REGION Network 60: ST04->ST05
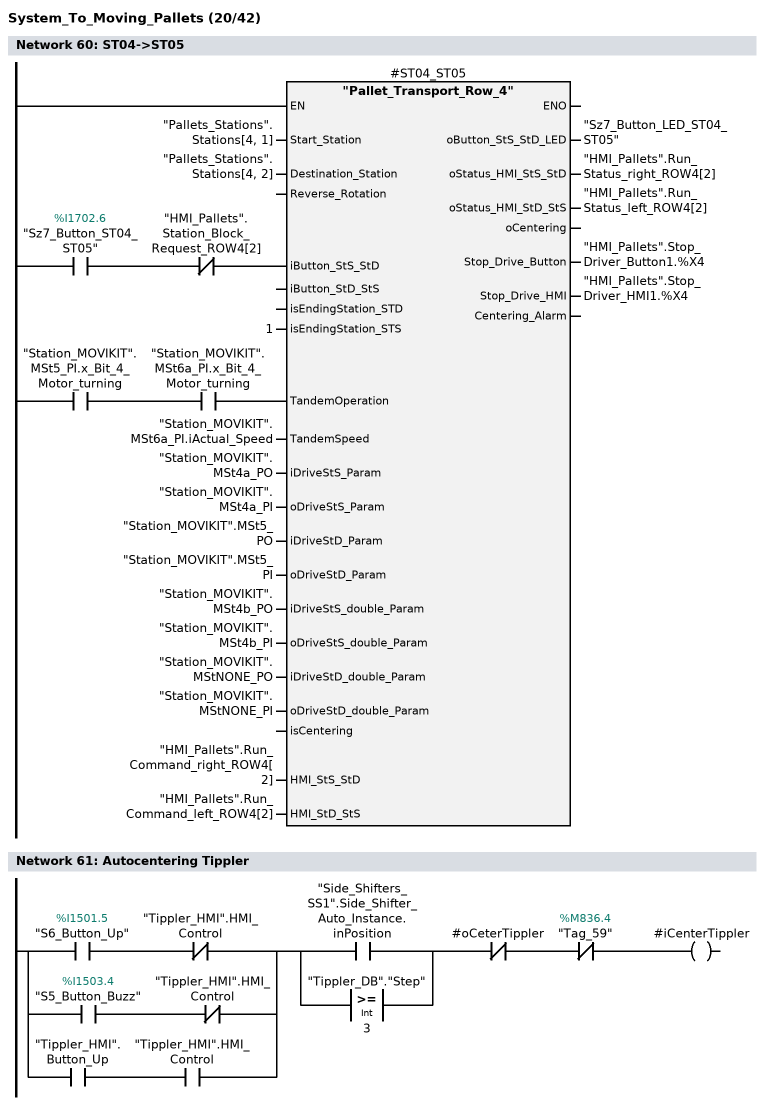
   RUNG wire#powerrail
      #ST04_ST05(iButton_StS_StD := wire#w1, TandemOperation := wire#w2, Start_Station := "Pallets_Stations".Stations[4, 1], Destination_Station := "Pallets_Stations".Stations[4, 2], Reverse_Rotation :=, iButton_StD_StS :=, isEndingStation_STD :=, isEndingStation_STS := 1, TandemSpeed := "Station_MOVIKIT".MSt6a_PI.iActual_Speed, iDriveStS_Param := "Station_MOVIKIT".MSt4a_PO, oDriveStS_Param := "Station_MOVIKIT".MSt4a_PI, iDriveStD_Param := "Station_MOVIKIT".MSt5_PO, oDriveStD_Param := "Station_MOVIKIT".MSt5_PI, iDriveStS_double_Param := "Station_MOVIKIT".MSt4b_PO, oDriveStS_double_Param := "Station_MOVIKIT".MSt4b_PI, iDriveStD_double_Param := "Station_MOVIKIT".MStNONE_PO, oDriveStD_double_Param := "Station_MOVIKIT".MStNONE_PI, isCentering :=, HMI_StS_StD := "HMI_Pallets".Run_Command_right_ROW4[2], HMI_StD_StS := "HMI_Pallets".Run_Command_left_ROW4[2], oButton_StS_StD_LED => "Sz7_Button_LED_ST04_ST05", oStatus_HMI_StS_StD => "HMI_Pallets".Run_Status_right_ROW4[2], oStatus_HMI_StD_StS => "HMI_Pallets".Run_Status_left_ROW4[2], oCentering =>, Stop_Drive_Button => "HMI_Pallets".Stop_Driver_Button1.%X4, Stop_Drive_HMI => "HMI_Pallets".Stop_Driver_HMI1.%X4, Centering_Alarm =>)
   END_RUNG
   RUNG wire#powerrail
      Contact( "Sz7_Button_ST04_ST05" )
      I_Contact( "HMI_Pallets".Station_Block_Request_ROW4[2] )
   END_RUNG wire#w1
   RUNG wire#powerrail
      Contact( "Station_MOVIKIT".MSt5_PI.x_Bit_4_Motor_turning )
      Contact( "Station_MOVIKIT".MSt6a_PI.x_Bit_4_Motor_turning )
   END_RUNG wire#w2
   // the same network as SCL:
   #ST04_ST05(Start_Station := "Pallets_Stations".Stations[4, 1],   // "Pallet_Transport_Row_4"
              Destination_Station := "Pallets_Stations".Stations[4, 2],
              iButton_StS_StD := "Sz7_Button_ST04_ST05" AND NOT "HMI_Pallets".Station_Block_Request_ROW4[2],
              isEndingStation_STS := 1,
              TandemOperation := "Station_MOVIKIT".MSt5_PI.x_Bit_4_Motor_turning AND "Station_MOVIKIT".MSt6a_PI.x_Bit_4_Motor_turning,
              TandemSpeed := "Station_MOVIKIT".MSt6a_PI.iActual_Speed,
              iDriveStS_Param := "Station_MOVIKIT".MSt4a_PO,
              oDriveStS_Param := "Station_MOVIKIT".MSt4a_PI,
              iDriveStD_Param := "Station_MOVIKIT".MSt5_PO,
              oDriveStD_Param := "Station_MOVIKIT".MSt5_PI,
              iDriveStS_double_Param := "Station_MOVIKIT".MSt4b_PO,
              oDriveStS_double_Param := "Station_MOVIKIT".MSt4b_PI,
              iDriveStD_double_Param := "Station_MOVIKIT".MStNONE_PO,
              oDriveStD_double_Param := "Station_MOVIKIT".MStNONE_PI,
              HMI_StS_StD := "HMI_Pallets".Run_Command_right_ROW4[2],
              HMI_StD_StS := "HMI_Pallets".Run_Command_left_ROW4[2],
              oButton_StS_StD_LED => "Sz7_Button_LED_ST04_ST05",
              oStatus_HMI_StS_StD => "HMI_Pallets".Run_Status_right_ROW4[2],
              oStatus_HMI_StD_StS => "HMI_Pallets".Run_Status_left_ROW4[2],
              Stop_Drive_Button => "HMI_Pallets".Stop_Driver_Button1.%X4,
              Stop_Drive_HMI => "HMI_Pallets".Stop_Driver_HMI1.%X4);
END_REGION

REGION Network 61: Autocentering Tippler
   RUNG wire#powerrail
      Contact( "S6_Button_Up" )
      I_Contact( "Tippler_HMI".HMI_Control )
      wire#w1
      Contact( "Side_Shifters_SS1".Side_Shifter_Auto_Instance.inPosition )
      wire#w2
      I_Contact( #oCeterTippler )
      I_Contact( "Tag_59" )
      Coil( #iCenterTippler )
   END_RUNG
   RUNG wire#powerrail
      Contact( "S5_Button_Buzz" )
      I_Contact( "Tippler_HMI".HMI_Control )
   END_RUNG wire#w1
   RUNG wire#powerrail
      Contact( "Tippler_HMI".Button_Up )
      Contact( "Tippler_HMI".HMI_Control )
   END_RUNG wire#w1
   RUNG wire#w1
      { S7_Templates := "SrcType := Int" } GE_Contact(in1 := "Tippler_DB"."Step", in2 := 3)
   END_RUNG wire#w2
   // the same network as SCL:
   #iCenterTippler := (("S6_Button_Up" AND NOT "Tippler_HMI".HMI_Control) OR ("S5_Button_Buzz" AND NOT "Tippler_HMI".HMI_Control) OR ("Tippler_HMI".Button_Up AND "Tippler_HMI".HMI_Control)) AND ("Side_Shifters_SS1".Side_Shifter_Auto_Instance.inPosition OR ("Tippler_DB"."Step" >= 3)) AND NOT #oCeterTippler AND NOT "Tag_59";
END_REGION

REGION Network 62: ST01->ST02
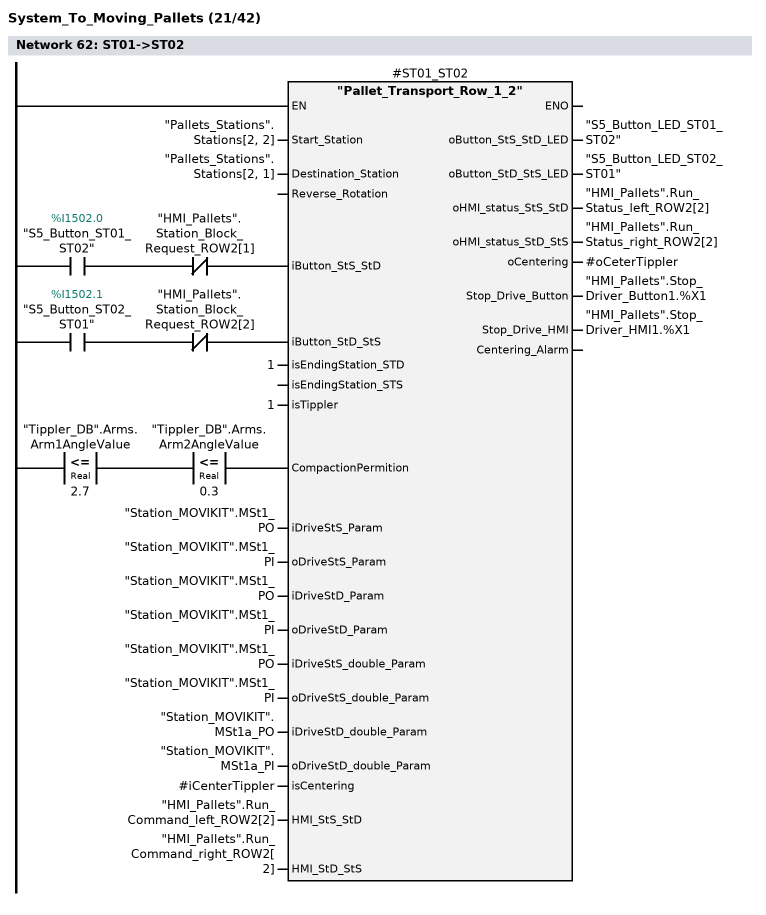
   RUNG wire#powerrail
      #ST01_ST02(iButton_StS_StD := wire#w1, iButton_StD_StS := wire#w2, CompactionPermition := wire#w3, Start_Station := "Pallets_Stations".Stations[2, 2], Destination_Station := "Pallets_Stations".Stations[2, 1], Reverse_Rotation :=, isEndingStation_STD := 1, isEndingStation_STS :=, isTippler := 1, iDriveStS_Param := "Station_MOVIKIT".MSt1_PO, oDriveStS_Param := "Station_MOVIKIT".MSt1_PI, iDriveStD_Param := "Station_MOVIKIT".MSt1_PO, oDriveStD_Param := "Station_MOVIKIT".MSt1_PI, iDriveStS_double_Param := "Station_MOVIKIT".MSt1_PO, oDriveStS_double_Param := "Station_MOVIKIT".MSt1_PI, iDriveStD_double_Param := "Station_MOVIKIT".MSt1a_PO, oDriveStD_double_Param := "Station_MOVIKIT".MSt1a_PI, isCentering := #iCenterTippler, HMI_StS_StD := "HMI_Pallets".Run_Command_left_ROW2[2], HMI_StD_StS := "HMI_Pallets".Run_Command_right_ROW2[2], oButton_StS_StD_LED => "S5_Button_LED_ST01_ST02", oButton_StD_StS_LED => "S5_Button_LED_ST02_ST01", oHMI_status_StS_StD => "HMI_Pallets".Run_Status_left_ROW2[2], oHMI_status_StD_StS => "HMI_Pallets".Run_Status_right_ROW2[2], oCentering => #oCeterTippler, Stop_Drive_Button => "HMI_Pallets".Stop_Driver_Button1.%X1, Stop_Drive_HMI => "HMI_Pallets".Stop_Driver_HMI1.%X1, Centering_Alarm =>)
   END_RUNG
   RUNG wire#powerrail
      Contact( "S5_Button_ST01_ST02" )
      I_Contact( "HMI_Pallets".Station_Block_Request_ROW2[1] )
   END_RUNG wire#w1
   RUNG wire#powerrail
      Contact( "S5_Button_ST02_ST01" )
      I_Contact( "HMI_Pallets".Station_Block_Request_ROW2[2] )
   END_RUNG wire#w2
   RUNG wire#powerrail
      { S7_Templates := "SrcType := Real" } LE_Contact(in1 := "Tippler_DB".Arms.Arm1AngleValue, in2 := 2.7)
      { S7_Templates := "SrcType := Real" } LE_Contact(in1 := "Tippler_DB".Arms.Arm2AngleValue, in2 := 0.3)
   END_RUNG wire#w3
   // the same network as SCL:
   #ST01_ST02(Start_Station := "Pallets_Stations".Stations[2, 2],   // "Pallet_Transport_Row_1_2"
              Destination_Station := "Pallets_Stations".Stations[2, 1],
              iButton_StS_StD := "S5_Button_ST01_ST02" AND NOT "HMI_Pallets".Station_Block_Request_ROW2[1],
              iButton_StD_StS := "S5_Button_ST02_ST01" AND NOT "HMI_Pallets".Station_Block_Request_ROW2[2],
              isEndingStation_STD := 1,
              isTippler := 1,
              CompactionPermition := ("Tippler_DB".Arms.Arm1AngleValue <= 2.7) AND ("Tippler_DB".Arms.Arm2AngleValue <= 0.3),
              iDriveStS_Param := "Station_MOVIKIT".MSt1_PO,
              oDriveStS_Param := "Station_MOVIKIT".MSt1_PI,
              iDriveStD_Param := "Station_MOVIKIT".MSt1_PO,
              oDriveStD_Param := "Station_MOVIKIT".MSt1_PI,
              iDriveStS_double_Param := "Station_MOVIKIT".MSt1_PO,
              oDriveStS_double_Param := "Station_MOVIKIT".MSt1_PI,
              iDriveStD_double_Param := "Station_MOVIKIT".MSt1a_PO,
              oDriveStD_double_Param := "Station_MOVIKIT".MSt1a_PI,
              isCentering := #iCenterTippler,
              HMI_StS_StD := "HMI_Pallets".Run_Command_left_ROW2[2],
              HMI_StD_StS := "HMI_Pallets".Run_Command_right_ROW2[2],
              oButton_StS_StD_LED => "S5_Button_LED_ST01_ST02",
              oButton_StD_StS_LED => "S5_Button_LED_ST02_ST01",
              oHMI_status_StS_StD => "HMI_Pallets".Run_Status_left_ROW2[2],
              oHMI_status_StD_StS => "HMI_Pallets".Run_Status_right_ROW2[2],
              oCentering => #oCeterTippler,
              Stop_Drive_Button => "HMI_Pallets".Stop_Driver_Button1.%X1,
              Stop_Drive_HMI => "HMI_Pallets".Stop_Driver_HMI1.%X1);
END_REGION

REGION Network 63: ST38->ST01
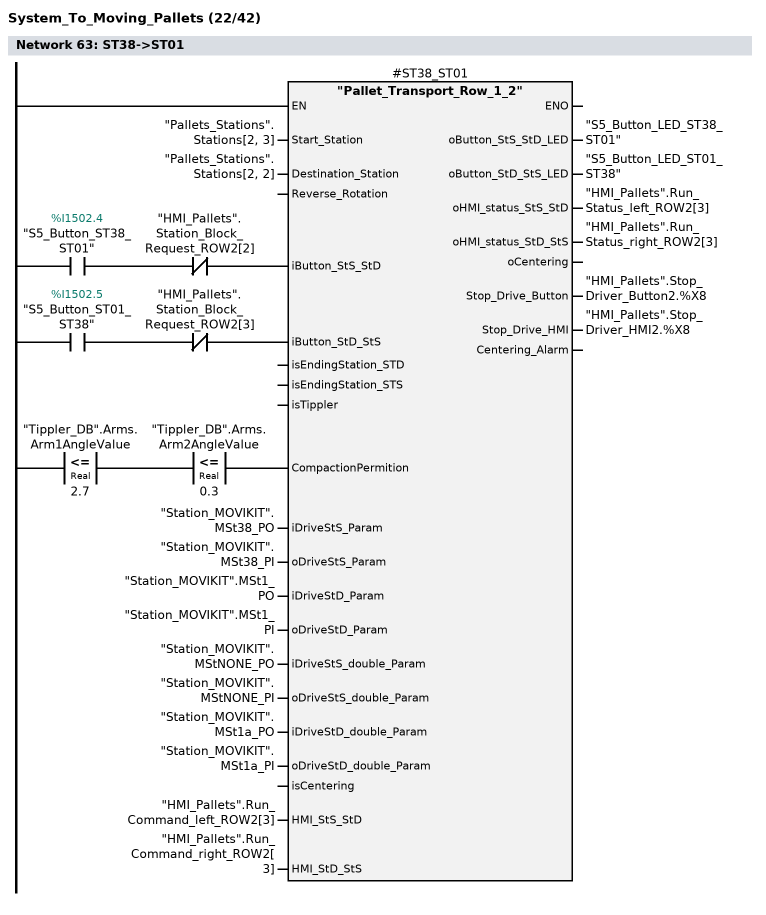
   RUNG wire#powerrail
      #ST38_ST01(iButton_StS_StD := wire#w1, iButton_StD_StS := wire#w2, CompactionPermition := wire#w3, Start_Station := "Pallets_Stations".Stations[2, 3], Destination_Station := "Pallets_Stations".Stations[2, 2], Reverse_Rotation :=, isEndingStation_STD :=, isEndingStation_STS :=, isTippler :=, iDriveStS_Param := "Station_MOVIKIT".MSt38_PO, oDriveStS_Param := "Station_MOVIKIT".MSt38_PI, iDriveStD_Param := "Station_MOVIKIT".MSt1_PO, oDriveStD_Param := "Station_MOVIKIT".MSt1_PI, iDriveStS_double_Param := "Station_MOVIKIT".MStNONE_PO, oDriveStS_double_Param := "Station_MOVIKIT".MStNONE_PI, iDriveStD_double_Param := "Station_MOVIKIT".MSt1a_PO, oDriveStD_double_Param := "Station_MOVIKIT".MSt1a_PI, isCentering :=, HMI_StS_StD := "HMI_Pallets".Run_Command_left_ROW2[3], HMI_StD_StS := "HMI_Pallets".Run_Command_right_ROW2[3], oButton_StS_StD_LED => "S5_Button_LED_ST38_ST01", oButton_StD_StS_LED => "S5_Button_LED_ST01_ST38", oHMI_status_StS_StD => "HMI_Pallets".Run_Status_left_ROW2[3], oHMI_status_StD_StS => "HMI_Pallets".Run_Status_right_ROW2[3], oCentering =>, Stop_Drive_Button => "HMI_Pallets".Stop_Driver_Button2.%X8, Stop_Drive_HMI => "HMI_Pallets".Stop_Driver_HMI2.%X8, Centering_Alarm =>)
   END_RUNG
   RUNG wire#powerrail
      Contact( "S5_Button_ST38_ST01" )
      I_Contact( "HMI_Pallets".Station_Block_Request_ROW2[2] )
   END_RUNG wire#w1
   RUNG wire#powerrail
      Contact( "S5_Button_ST01_ST38" )
      I_Contact( "HMI_Pallets".Station_Block_Request_ROW2[3] )
   END_RUNG wire#w2
   RUNG wire#powerrail
      { S7_Templates := "SrcType := Real" } LE_Contact(in1 := "Tippler_DB".Arms.Arm1AngleValue, in2 := 2.7)
      { S7_Templates := "SrcType := Real" } LE_Contact(in1 := "Tippler_DB".Arms.Arm2AngleValue, in2 := 0.3)
   END_RUNG wire#w3
   // the same network as SCL:
   #ST38_ST01(Start_Station := "Pallets_Stations".Stations[2, 3],   // "Pallet_Transport_Row_1_2"
              Destination_Station := "Pallets_Stations".Stations[2, 2],
              iButton_StS_StD := "S5_Button_ST38_ST01" AND NOT "HMI_Pallets".Station_Block_Request_ROW2[2],
              iButton_StD_StS := "S5_Button_ST01_ST38" AND NOT "HMI_Pallets".Station_Block_Request_ROW2[3],
              CompactionPermition := ("Tippler_DB".Arms.Arm1AngleValue <= 2.7) AND ("Tippler_DB".Arms.Arm2AngleValue <= 0.3),
              iDriveStS_Param := "Station_MOVIKIT".MSt38_PO,
              oDriveStS_Param := "Station_MOVIKIT".MSt38_PI,
              iDriveStD_Param := "Station_MOVIKIT".MSt1_PO,
              oDriveStD_Param := "Station_MOVIKIT".MSt1_PI,
              iDriveStS_double_Param := "Station_MOVIKIT".MStNONE_PO,
              oDriveStS_double_Param := "Station_MOVIKIT".MStNONE_PI,
              iDriveStD_double_Param := "Station_MOVIKIT".MSt1a_PO,
              oDriveStD_double_Param := "Station_MOVIKIT".MSt1a_PI,
              HMI_StS_StD := "HMI_Pallets".Run_Command_left_ROW2[3],
              HMI_StD_StS := "HMI_Pallets".Run_Command_right_ROW2[3],
              oButton_StS_StD_LED => "S5_Button_LED_ST38_ST01",
              oButton_StD_StS_LED => "S5_Button_LED_ST01_ST38",
              oHMI_status_StS_StD => "HMI_Pallets".Run_Status_left_ROW2[3],
              oHMI_status_StD_StS => "HMI_Pallets".Run_Status_right_ROW2[3],
              Stop_Drive_Button => "HMI_Pallets".Stop_Driver_Button2.%X8,
              Stop_Drive_HMI => "HMI_Pallets".Stop_Driver_HMI2.%X8);
END_REGION

REGION Network 64: ST34->ST35
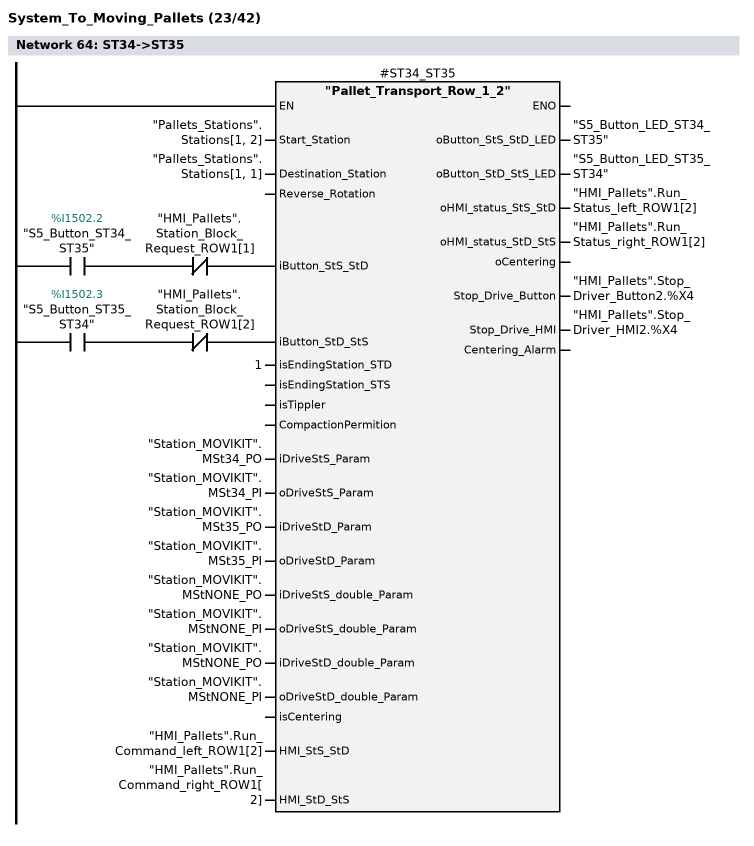
   RUNG wire#powerrail
      #ST34_ST35(iButton_StS_StD := wire#w1, iButton_StD_StS := wire#w2, Start_Station := "Pallets_Stations".Stations[1, 2], Destination_Station := "Pallets_Stations".Stations[1, 1], Reverse_Rotation :=, isEndingStation_STD := 1, isEndingStation_STS :=, isTippler :=, CompactionPermition :=, iDriveStS_Param := "Station_MOVIKIT".MSt34_PO, oDriveStS_Param := "Station_MOVIKIT".MSt34_PI, iDriveStD_Param := "Station_MOVIKIT".MSt35_PO, oDriveStD_Param := "Station_MOVIKIT".MSt35_PI, iDriveStS_double_Param := "Station_MOVIKIT".MStNONE_PO, oDriveStS_double_Param := "Station_MOVIKIT".MStNONE_PI, iDriveStD_double_Param := "Station_MOVIKIT".MStNONE_PO, oDriveStD_double_Param := "Station_MOVIKIT".MStNONE_PI, isCentering :=, HMI_StS_StD := "HMI_Pallets".Run_Command_left_ROW1[2], HMI_StD_StS := "HMI_Pallets".Run_Command_right_ROW1[2], oButton_StS_StD_LED => "S5_Button_LED_ST34_ST35", oButton_StD_StS_LED => "S5_Button_LED_ST35_ST34", oHMI_status_StS_StD => "HMI_Pallets".Run_Status_left_ROW1[2], oHMI_status_StD_StS => "HMI_Pallets".Run_Status_right_ROW1[2], oCentering =>, Stop_Drive_Button => "HMI_Pallets".Stop_Driver_Button2.%X4, Stop_Drive_HMI => "HMI_Pallets".Stop_Driver_HMI2.%X4, Centering_Alarm =>)
   END_RUNG
   RUNG wire#powerrail
      Contact( "S5_Button_ST34_ST35" )
      I_Contact( "HMI_Pallets".Station_Block_Request_ROW1[1] )
   END_RUNG wire#w1
   RUNG wire#powerrail
      Contact( "S5_Button_ST35_ST34" )
      I_Contact( "HMI_Pallets".Station_Block_Request_ROW1[2] )
   END_RUNG wire#w2
   // the same network as SCL:
   #ST34_ST35(Start_Station := "Pallets_Stations".Stations[1, 2],   // "Pallet_Transport_Row_1_2"
              Destination_Station := "Pallets_Stations".Stations[1, 1],
              iButton_StS_StD := "S5_Button_ST34_ST35" AND NOT "HMI_Pallets".Station_Block_Request_ROW1[1],
              iButton_StD_StS := "S5_Button_ST35_ST34" AND NOT "HMI_Pallets".Station_Block_Request_ROW1[2],
              isEndingStation_STD := 1,
              iDriveStS_Param := "Station_MOVIKIT".MSt34_PO,
              oDriveStS_Param := "Station_MOVIKIT".MSt34_PI,
              iDriveStD_Param := "Station_MOVIKIT".MSt35_PO,
              oDriveStD_Param := "Station_MOVIKIT".MSt35_PI,
              iDriveStS_double_Param := "Station_MOVIKIT".MStNONE_PO,
              oDriveStS_double_Param := "Station_MOVIKIT".MStNONE_PI,
              iDriveStD_double_Param := "Station_MOVIKIT".MStNONE_PO,
              oDriveStD_double_Param := "Station_MOVIKIT".MStNONE_PI,
              HMI_StS_StD := "HMI_Pallets".Run_Command_left_ROW1[2],
              HMI_StD_StS := "HMI_Pallets".Run_Command_right_ROW1[2],
              oButton_StS_StD_LED => "S5_Button_LED_ST34_ST35",
              oButton_StD_StS_LED => "S5_Button_LED_ST35_ST34",
              oHMI_status_StS_StD => "HMI_Pallets".Run_Status_left_ROW1[2],
              oHMI_status_StD_StS => "HMI_Pallets".Run_Status_right_ROW1[2],
              Stop_Drive_Button => "HMI_Pallets".Stop_Driver_Button2.%X4,
              Stop_Drive_HMI => "HMI_Pallets".Stop_Driver_HMI2.%X4);
END_REGION

REGION Network 65: ST33->ST34
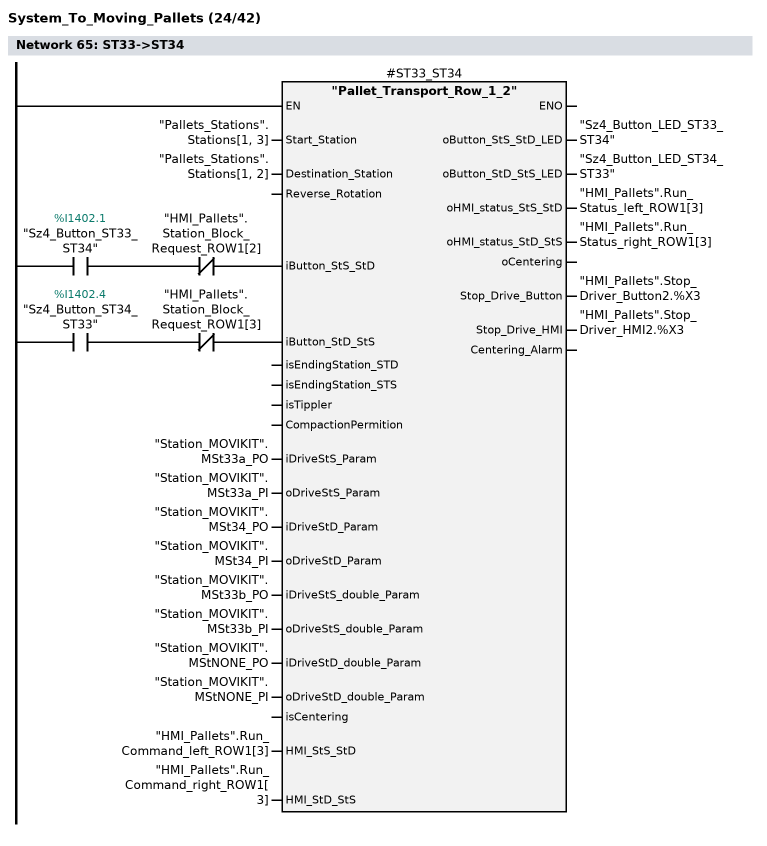
   RUNG wire#powerrail
      #ST33_ST34(iButton_StS_StD := wire#w1, iButton_StD_StS := wire#w2, Start_Station := "Pallets_Stations".Stations[1, 3], Destination_Station := "Pallets_Stations".Stations[1, 2], Reverse_Rotation :=, isEndingStation_STD :=, isEndingStation_STS :=, isTippler :=, CompactionPermition :=, iDriveStS_Param := "Station_MOVIKIT".MSt33a_PO, oDriveStS_Param := "Station_MOVIKIT".MSt33a_PI, iDriveStD_Param := "Station_MOVIKIT".MSt34_PO, oDriveStD_Param := "Station_MOVIKIT".MSt34_PI, iDriveStS_double_Param := "Station_MOVIKIT".MSt33b_PO, oDriveStS_double_Param := "Station_MOVIKIT".MSt33b_PI, iDriveStD_double_Param := "Station_MOVIKIT".MStNONE_PO, oDriveStD_double_Param := "Station_MOVIKIT".MStNONE_PI, isCentering :=, HMI_StS_StD := "HMI_Pallets".Run_Command_left_ROW1[3], HMI_StD_StS := "HMI_Pallets".Run_Command_right_ROW1[3], oButton_StS_StD_LED => "Sz4_Button_LED_ST33_ST34", oButton_StD_StS_LED => "Sz4_Button_LED_ST34_ST33", oHMI_status_StS_StD => "HMI_Pallets".Run_Status_left_ROW1[3], oHMI_status_StD_StS => "HMI_Pallets".Run_Status_right_ROW1[3], oCentering =>, Stop_Drive_Button => "HMI_Pallets".Stop_Driver_Button2.%X3, Stop_Drive_HMI => "HMI_Pallets".Stop_Driver_HMI2.%X3, Centering_Alarm =>)
   END_RUNG
   RUNG wire#powerrail
      Contact( "Sz4_Button_ST33_ST34" )
      I_Contact( "HMI_Pallets".Station_Block_Request_ROW1[2] )
   END_RUNG wire#w1
   RUNG wire#powerrail
      Contact( "Sz4_Button_ST34_ST33" )
      I_Contact( "HMI_Pallets".Station_Block_Request_ROW1[3] )
   END_RUNG wire#w2
   // the same network as SCL:
   #ST33_ST34(Start_Station := "Pallets_Stations".Stations[1, 3],   // "Pallet_Transport_Row_1_2"
              Destination_Station := "Pallets_Stations".Stations[1, 2],
              iButton_StS_StD := "Sz4_Button_ST33_ST34" AND NOT "HMI_Pallets".Station_Block_Request_ROW1[2],
              iButton_StD_StS := "Sz4_Button_ST34_ST33" AND NOT "HMI_Pallets".Station_Block_Request_ROW1[3],
              iDriveStS_Param := "Station_MOVIKIT".MSt33a_PO,
              oDriveStS_Param := "Station_MOVIKIT".MSt33a_PI,
              iDriveStD_Param := "Station_MOVIKIT".MSt34_PO,
              oDriveStD_Param := "Station_MOVIKIT".MSt34_PI,
              iDriveStS_double_Param := "Station_MOVIKIT".MSt33b_PO,
              oDriveStS_double_Param := "Station_MOVIKIT".MSt33b_PI,
              iDriveStD_double_Param := "Station_MOVIKIT".MStNONE_PO,
              oDriveStD_double_Param := "Station_MOVIKIT".MStNONE_PI,
              HMI_StS_StD := "HMI_Pallets".Run_Command_left_ROW1[3],
              HMI_StD_StS := "HMI_Pallets".Run_Command_right_ROW1[3],
              oButton_StS_StD_LED => "Sz4_Button_LED_ST33_ST34",
              oButton_StD_StS_LED => "Sz4_Button_LED_ST34_ST33",
              oHMI_status_StS_StD => "HMI_Pallets".Run_Status_left_ROW1[3],
              oHMI_status_StD_StS => "HMI_Pallets".Run_Status_right_ROW1[3],
              Stop_Drive_Button => "HMI_Pallets".Stop_Driver_Button2.%X3,
              Stop_Drive_HMI => "HMI_Pallets".Stop_Driver_HMI2.%X3);
END_REGION

REGION Network 66: ST32->ST33
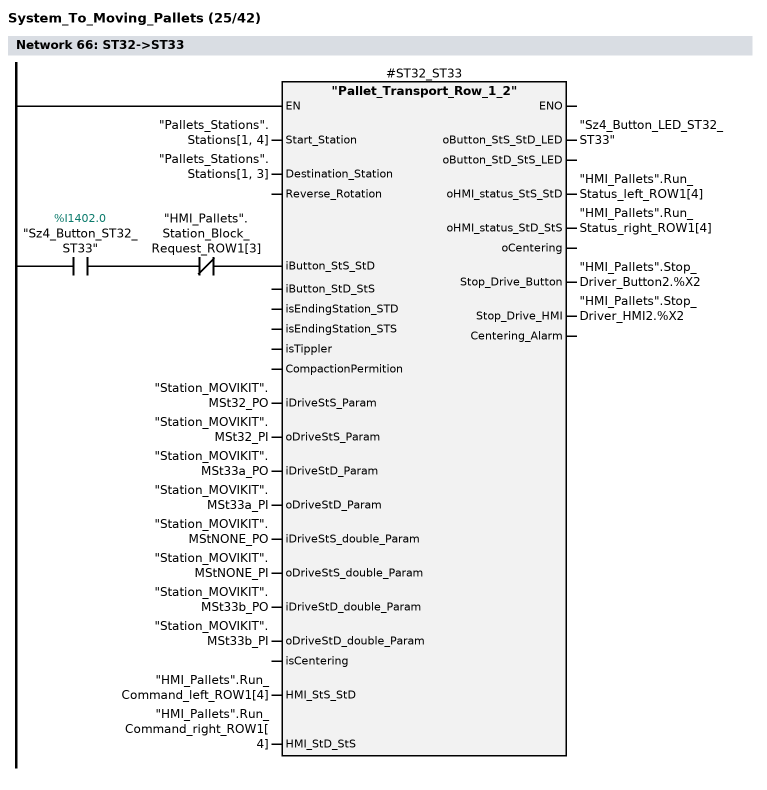
   RUNG wire#powerrail
      #ST32_ST33(iButton_StS_StD := wire#w1, Start_Station := "Pallets_Stations".Stations[1, 4], Destination_Station := "Pallets_Stations".Stations[1, 3], Reverse_Rotation :=, iButton_StD_StS :=, isEndingStation_STD :=, isEndingStation_STS :=, isTippler :=, CompactionPermition :=, iDriveStS_Param := "Station_MOVIKIT".MSt32_PO, oDriveStS_Param := "Station_MOVIKIT".MSt32_PI, iDriveStD_Param := "Station_MOVIKIT".MSt33a_PO, oDriveStD_Param := "Station_MOVIKIT".MSt33a_PI, iDriveStS_double_Param := "Station_MOVIKIT".MStNONE_PO, oDriveStS_double_Param := "Station_MOVIKIT".MStNONE_PI, iDriveStD_double_Param := "Station_MOVIKIT".MSt33b_PO, oDriveStD_double_Param := "Station_MOVIKIT".MSt33b_PI, isCentering :=, HMI_StS_StD := "HMI_Pallets".Run_Command_left_ROW1[4], HMI_StD_StS := "HMI_Pallets".Run_Command_right_ROW1[4], oButton_StS_StD_LED => "Sz4_Button_LED_ST32_ST33", oButton_StD_StS_LED =>, oHMI_status_StS_StD => "HMI_Pallets".Run_Status_left_ROW1[4], oHMI_status_StD_StS => "HMI_Pallets".Run_Status_right_ROW1[4], oCentering =>, Stop_Drive_Button => "HMI_Pallets".Stop_Driver_Button2.%X2, Stop_Drive_HMI => "HMI_Pallets".Stop_Driver_HMI2.%X2, Centering_Alarm =>)
   END_RUNG
   RUNG wire#powerrail
      Contact( "Sz4_Button_ST32_ST33" )
      I_Contact( "HMI_Pallets".Station_Block_Request_ROW1[3] )
   END_RUNG wire#w1
   // the same network as SCL:
   #ST32_ST33(Start_Station := "Pallets_Stations".Stations[1, 4],   // "Pallet_Transport_Row_1_2"
              Destination_Station := "Pallets_Stations".Stations[1, 3],
              iButton_StS_StD := "Sz4_Button_ST32_ST33" AND NOT "HMI_Pallets".Station_Block_Request_ROW1[3],
              iDriveStS_Param := "Station_MOVIKIT".MSt32_PO,
              oDriveStS_Param := "Station_MOVIKIT".MSt32_PI,
              iDriveStD_Param := "Station_MOVIKIT".MSt33a_PO,
              oDriveStD_Param := "Station_MOVIKIT".MSt33a_PI,
              iDriveStS_double_Param := "Station_MOVIKIT".MStNONE_PO,
              oDriveStS_double_Param := "Station_MOVIKIT".MStNONE_PI,
              iDriveStD_double_Param := "Station_MOVIKIT".MSt33b_PO,
              oDriveStD_double_Param := "Station_MOVIKIT".MSt33b_PI,
              HMI_StS_StD := "HMI_Pallets".Run_Command_left_ROW1[4],
              HMI_StD_StS := "HMI_Pallets".Run_Command_right_ROW1[4],
              oButton_StS_StD_LED => "Sz4_Button_LED_ST32_ST33",
              oHMI_status_StS_StD => "HMI_Pallets".Run_Status_left_ROW1[4],
              oHMI_status_StD_StS => "HMI_Pallets".Run_Status_right_ROW1[4],
              Stop_Drive_Button => "HMI_Pallets".Stop_Driver_Button2.%X2,
              Stop_Drive_HMI => "HMI_Pallets".Stop_Driver_HMI2.%X2);
END_REGION

REGION Network 67: ST31->ST32
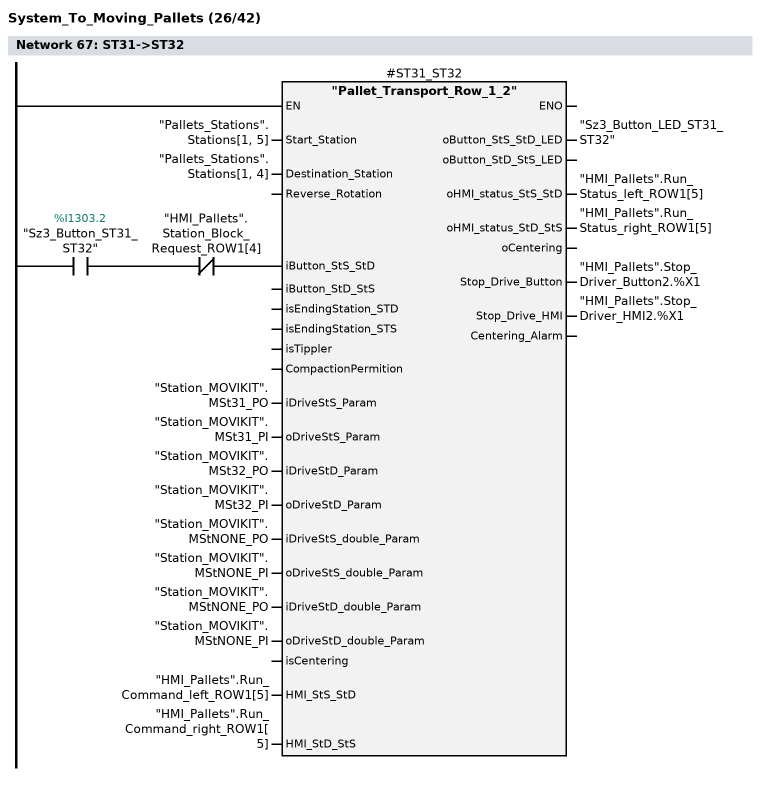
   RUNG wire#powerrail
      #ST31_ST32(iButton_StS_StD := wire#w1, Start_Station := "Pallets_Stations".Stations[1, 5], Destination_Station := "Pallets_Stations".Stations[1, 4], Reverse_Rotation :=, iButton_StD_StS :=, isEndingStation_STD :=, isEndingStation_STS :=, isTippler :=, CompactionPermition :=, iDriveStS_Param := "Station_MOVIKIT".MSt31_PO, oDriveStS_Param := "Station_MOVIKIT".MSt31_PI, iDriveStD_Param := "Station_MOVIKIT".MSt32_PO, oDriveStD_Param := "Station_MOVIKIT".MSt32_PI, iDriveStS_double_Param := "Station_MOVIKIT".MStNONE_PO, oDriveStS_double_Param := "Station_MOVIKIT".MStNONE_PI, iDriveStD_double_Param := "Station_MOVIKIT".MStNONE_PO, oDriveStD_double_Param := "Station_MOVIKIT".MStNONE_PI, isCentering :=, HMI_StS_StD := "HMI_Pallets".Run_Command_left_ROW1[5], HMI_StD_StS := "HMI_Pallets".Run_Command_right_ROW1[5], oButton_StS_StD_LED => "Sz3_Button_LED_ST31_ST32", oButton_StD_StS_LED =>, oHMI_status_StS_StD => "HMI_Pallets".Run_Status_left_ROW1[5], oHMI_status_StD_StS => "HMI_Pallets".Run_Status_right_ROW1[5], oCentering =>, Stop_Drive_Button => "HMI_Pallets".Stop_Driver_Button2.%X1, Stop_Drive_HMI => "HMI_Pallets".Stop_Driver_HMI2.%X1, Centering_Alarm =>)
   END_RUNG
   RUNG wire#powerrail
      Contact( "Sz3_Button_ST31_ST32" )
      I_Contact( "HMI_Pallets".Station_Block_Request_ROW1[4] )
   END_RUNG wire#w1
   // the same network as SCL:
   #ST31_ST32(Start_Station := "Pallets_Stations".Stations[1, 5],   // "Pallet_Transport_Row_1_2"
              Destination_Station := "Pallets_Stations".Stations[1, 4],
              iButton_StS_StD := "Sz3_Button_ST31_ST32" AND NOT "HMI_Pallets".Station_Block_Request_ROW1[4],
              iDriveStS_Param := "Station_MOVIKIT".MSt31_PO,
              oDriveStS_Param := "Station_MOVIKIT".MSt31_PI,
              iDriveStD_Param := "Station_MOVIKIT".MSt32_PO,
              oDriveStD_Param := "Station_MOVIKIT".MSt32_PI,
              iDriveStS_double_Param := "Station_MOVIKIT".MStNONE_PO,
              oDriveStS_double_Param := "Station_MOVIKIT".MStNONE_PI,
              iDriveStD_double_Param := "Station_MOVIKIT".MStNONE_PO,
              oDriveStD_double_Param := "Station_MOVIKIT".MStNONE_PI,
              HMI_StS_StD := "HMI_Pallets".Run_Command_left_ROW1[5],
              HMI_StD_StS := "HMI_Pallets".Run_Command_right_ROW1[5],
              oButton_StS_StD_LED => "Sz3_Button_LED_ST31_ST32",
              oHMI_status_StS_StD => "HMI_Pallets".Run_Status_left_ROW1[5],
              oHMI_status_StD_StS => "HMI_Pallets".Run_Status_right_ROW1[5],
              Stop_Drive_Button => "HMI_Pallets".Stop_Driver_Button2.%X1,
              Stop_Drive_HMI => "HMI_Pallets".Stop_Driver_HMI2.%X1);
END_REGION

REGION Network 68: ST30->ST31
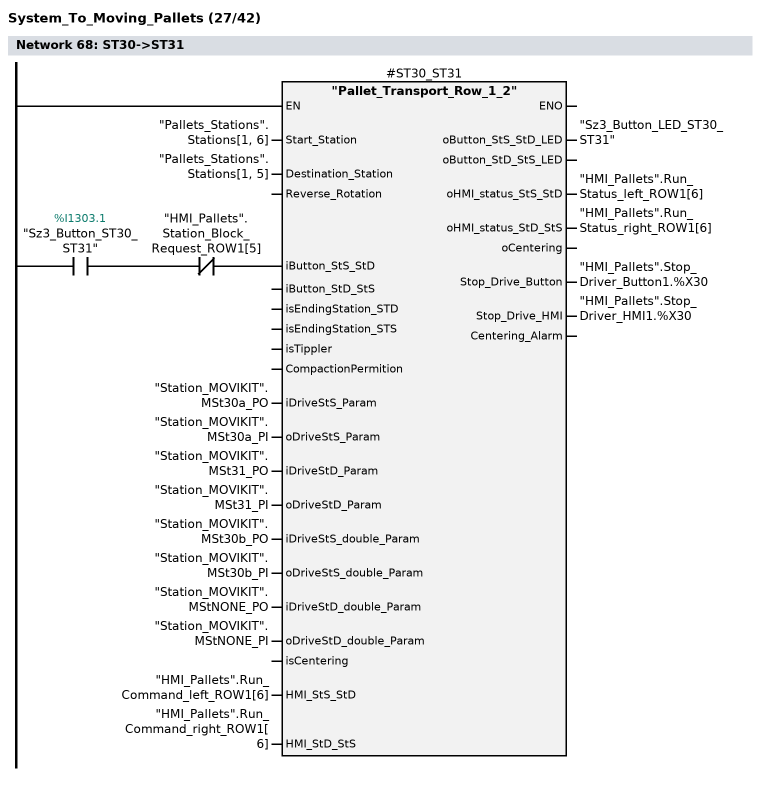
   RUNG wire#powerrail
      #ST30_ST31(iButton_StS_StD := wire#w1, Start_Station := "Pallets_Stations".Stations[1, 6], Destination_Station := "Pallets_Stations".Stations[1, 5], Reverse_Rotation :=, iButton_StD_StS :=, isEndingStation_STD :=, isEndingStation_STS :=, isTippler :=, CompactionPermition :=, iDriveStS_Param := "Station_MOVIKIT".MSt30a_PO, oDriveStS_Param := "Station_MOVIKIT".MSt30a_PI, iDriveStD_Param := "Station_MOVIKIT".MSt31_PO, oDriveStD_Param := "Station_MOVIKIT".MSt31_PI, iDriveStS_double_Param := "Station_MOVIKIT".MSt30b_PO, oDriveStS_double_Param := "Station_MOVIKIT".MSt30b_PI, iDriveStD_double_Param := "Station_MOVIKIT".MStNONE_PO, oDriveStD_double_Param := "Station_MOVIKIT".MStNONE_PI, isCentering :=, HMI_StS_StD := "HMI_Pallets".Run_Command_left_ROW1[6], HMI_StD_StS := "HMI_Pallets".Run_Command_right_ROW1[6], oButton_StS_StD_LED => "Sz3_Button_LED_ST30_ST31", oButton_StD_StS_LED =>, oHMI_status_StS_StD => "HMI_Pallets".Run_Status_left_ROW1[6], oHMI_status_StD_StS => "HMI_Pallets".Run_Status_right_ROW1[6], oCentering =>, Stop_Drive_Button => "HMI_Pallets".Stop_Driver_Button1.%X30, Stop_Drive_HMI => "HMI_Pallets".Stop_Driver_HMI1.%X30, Centering_Alarm =>)
   END_RUNG
   RUNG wire#powerrail
      Contact( "Sz3_Button_ST30_ST31" )
      I_Contact( "HMI_Pallets".Station_Block_Request_ROW1[5] )
   END_RUNG wire#w1
   // the same network as SCL:
   #ST30_ST31(Start_Station := "Pallets_Stations".Stations[1, 6],   // "Pallet_Transport_Row_1_2"
              Destination_Station := "Pallets_Stations".Stations[1, 5],
              iButton_StS_StD := "Sz3_Button_ST30_ST31" AND NOT "HMI_Pallets".Station_Block_Request_ROW1[5],
              iDriveStS_Param := "Station_MOVIKIT".MSt30a_PO,
              oDriveStS_Param := "Station_MOVIKIT".MSt30a_PI,
              iDriveStD_Param := "Station_MOVIKIT".MSt31_PO,
              oDriveStD_Param := "Station_MOVIKIT".MSt31_PI,
              iDriveStS_double_Param := "Station_MOVIKIT".MSt30b_PO,
              oDriveStS_double_Param := "Station_MOVIKIT".MSt30b_PI,
              iDriveStD_double_Param := "Station_MOVIKIT".MStNONE_PO,
              oDriveStD_double_Param := "Station_MOVIKIT".MStNONE_PI,
              HMI_StS_StD := "HMI_Pallets".Run_Command_left_ROW1[6],
              HMI_StD_StS := "HMI_Pallets".Run_Command_right_ROW1[6],
              oButton_StS_StD_LED => "Sz3_Button_LED_ST30_ST31",
              oHMI_status_StS_StD => "HMI_Pallets".Run_Status_left_ROW1[6],
              oHMI_status_StD_StS => "HMI_Pallets".Run_Status_right_ROW1[6],
              Stop_Drive_Button => "HMI_Pallets".Stop_Driver_Button1.%X30,
              Stop_Drive_HMI => "HMI_Pallets".Stop_Driver_HMI1.%X30);
END_REGION

REGION Network 69: ST29->ST30
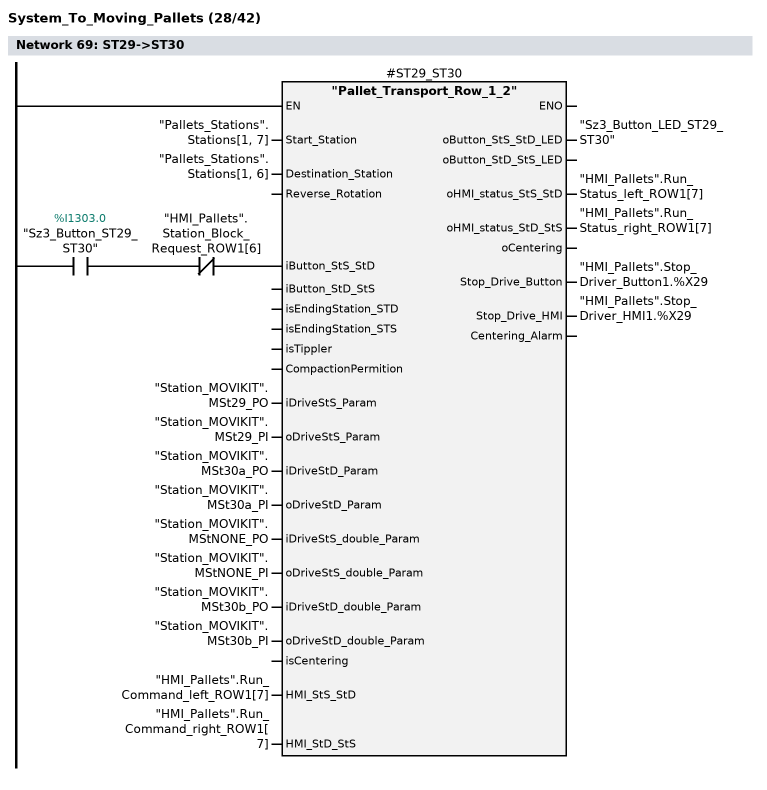
   RUNG wire#powerrail
      #ST29_ST30(iButton_StS_StD := wire#w1, Start_Station := "Pallets_Stations".Stations[1, 7], Destination_Station := "Pallets_Stations".Stations[1, 6], Reverse_Rotation :=, iButton_StD_StS :=, isEndingStation_STD :=, isEndingStation_STS :=, isTippler :=, CompactionPermition :=, iDriveStS_Param := "Station_MOVIKIT".MSt29_PO, oDriveStS_Param := "Station_MOVIKIT".MSt29_PI, iDriveStD_Param := "Station_MOVIKIT".MSt30a_PO, oDriveStD_Param := "Station_MOVIKIT".MSt30a_PI, iDriveStS_double_Param := "Station_MOVIKIT".MStNONE_PO, oDriveStS_double_Param := "Station_MOVIKIT".MStNONE_PI, iDriveStD_double_Param := "Station_MOVIKIT".MSt30b_PO, oDriveStD_double_Param := "Station_MOVIKIT".MSt30b_PI, isCentering :=, HMI_StS_StD := "HMI_Pallets".Run_Command_left_ROW1[7], HMI_StD_StS := "HMI_Pallets".Run_Command_right_ROW1[7], oButton_StS_StD_LED => "Sz3_Button_LED_ST29_ST30", oButton_StD_StS_LED =>, oHMI_status_StS_StD => "HMI_Pallets".Run_Status_left_ROW1[7], oHMI_status_StD_StS => "HMI_Pallets".Run_Status_right_ROW1[7], oCentering =>, Stop_Drive_Button => "HMI_Pallets".Stop_Driver_Button1.%X29, Stop_Drive_HMI => "HMI_Pallets".Stop_Driver_HMI1.%X29, Centering_Alarm =>)
   END_RUNG
   RUNG wire#powerrail
      Contact( "Sz3_Button_ST29_ST30" )
      I_Contact( "HMI_Pallets".Station_Block_Request_ROW1[6] )
   END_RUNG wire#w1
   // the same network as SCL:
   #ST29_ST30(Start_Station := "Pallets_Stations".Stations[1, 7],   // "Pallet_Transport_Row_1_2"
              Destination_Station := "Pallets_Stations".Stations[1, 6],
              iButton_StS_StD := "Sz3_Button_ST29_ST30" AND NOT "HMI_Pallets".Station_Block_Request_ROW1[6],
              iDriveStS_Param := "Station_MOVIKIT".MSt29_PO,
              oDriveStS_Param := "Station_MOVIKIT".MSt29_PI,
              iDriveStD_Param := "Station_MOVIKIT".MSt30a_PO,
              oDriveStD_Param := "Station_MOVIKIT".MSt30a_PI,
              iDriveStS_double_Param := "Station_MOVIKIT".MStNONE_PO,
              oDriveStS_double_Param := "Station_MOVIKIT".MStNONE_PI,
              iDriveStD_double_Param := "Station_MOVIKIT".MSt30b_PO,
              oDriveStD_double_Param := "Station_MOVIKIT".MSt30b_PI,
              HMI_StS_StD := "HMI_Pallets".Run_Command_left_ROW1[7],
              HMI_StD_StS := "HMI_Pallets".Run_Command_right_ROW1[7],
              oButton_StS_StD_LED => "Sz3_Button_LED_ST29_ST30",
              oHMI_status_StS_StD => "HMI_Pallets".Run_Status_left_ROW1[7],
              oHMI_status_StD_StS => "HMI_Pallets".Run_Status_right_ROW1[7],
              Stop_Drive_Button => "HMI_Pallets".Stop_Driver_Button1.%X29,
              Stop_Drive_HMI => "HMI_Pallets".Stop_Driver_HMI1.%X29);
END_REGION

REGION Network 70: ST28->ST29
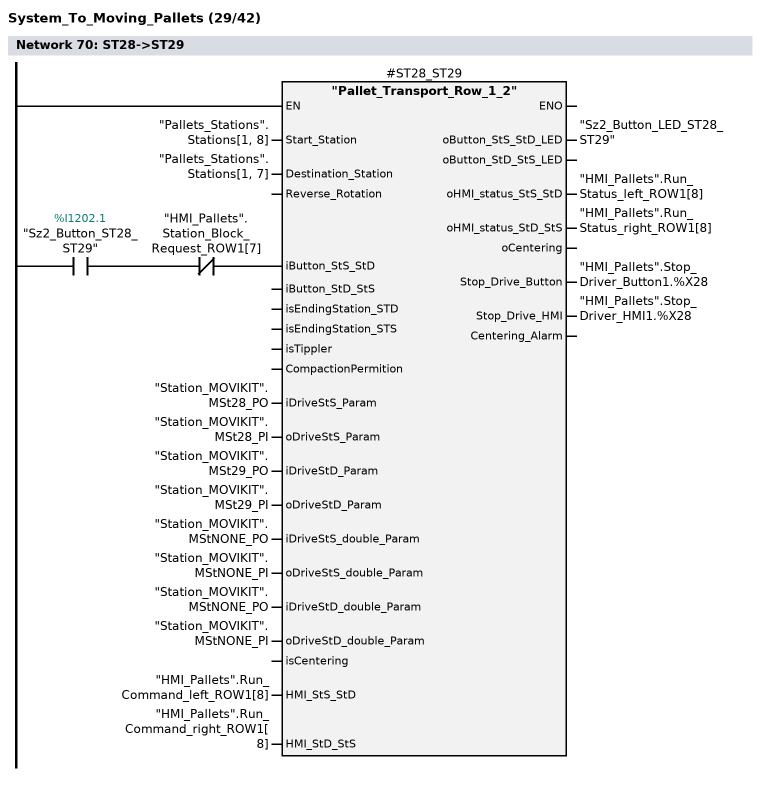
   RUNG wire#powerrail
      #ST28_ST29(iButton_StS_StD := wire#w1, Start_Station := "Pallets_Stations".Stations[1, 8], Destination_Station := "Pallets_Stations".Stations[1, 7], Reverse_Rotation :=, iButton_StD_StS :=, isEndingStation_STD :=, isEndingStation_STS :=, isTippler :=, CompactionPermition :=, iDriveStS_Param := "Station_MOVIKIT".MSt28_PO, oDriveStS_Param := "Station_MOVIKIT".MSt28_PI, iDriveStD_Param := "Station_MOVIKIT".MSt29_PO, oDriveStD_Param := "Station_MOVIKIT".MSt29_PI, iDriveStS_double_Param := "Station_MOVIKIT".MStNONE_PO, oDriveStS_double_Param := "Station_MOVIKIT".MStNONE_PI, iDriveStD_double_Param := "Station_MOVIKIT".MStNONE_PO, oDriveStD_double_Param := "Station_MOVIKIT".MStNONE_PI, isCentering :=, HMI_StS_StD := "HMI_Pallets".Run_Command_left_ROW1[8], HMI_StD_StS := "HMI_Pallets".Run_Command_right_ROW1[8], oButton_StS_StD_LED => "Sz2_Button_LED_ST28_ST29", oButton_StD_StS_LED =>, oHMI_status_StS_StD => "HMI_Pallets".Run_Status_left_ROW1[8], oHMI_status_StD_StS => "HMI_Pallets".Run_Status_right_ROW1[8], oCentering =>, Stop_Drive_Button => "HMI_Pallets".Stop_Driver_Button1.%X28, Stop_Drive_HMI => "HMI_Pallets".Stop_Driver_HMI1.%X28, Centering_Alarm =>)
   END_RUNG
   RUNG wire#powerrail
      Contact( "Sz2_Button_ST28_ST29" )
      I_Contact( "HMI_Pallets".Station_Block_Request_ROW1[7] )
   END_RUNG wire#w1
   // the same network as SCL:
   #ST28_ST29(Start_Station := "Pallets_Stations".Stations[1, 8],   // "Pallet_Transport_Row_1_2"
              Destination_Station := "Pallets_Stations".Stations[1, 7],
              iButton_StS_StD := "Sz2_Button_ST28_ST29" AND NOT "HMI_Pallets".Station_Block_Request_ROW1[7],
              iDriveStS_Param := "Station_MOVIKIT".MSt28_PO,
              oDriveStS_Param := "Station_MOVIKIT".MSt28_PI,
              iDriveStD_Param := "Station_MOVIKIT".MSt29_PO,
              oDriveStD_Param := "Station_MOVIKIT".MSt29_PI,
              iDriveStS_double_Param := "Station_MOVIKIT".MStNONE_PO,
              oDriveStS_double_Param := "Station_MOVIKIT".MStNONE_PI,
              iDriveStD_double_Param := "Station_MOVIKIT".MStNONE_PO,
              oDriveStD_double_Param := "Station_MOVIKIT".MStNONE_PI,
              HMI_StS_StD := "HMI_Pallets".Run_Command_left_ROW1[8],
              HMI_StD_StS := "HMI_Pallets".Run_Command_right_ROW1[8],
              oButton_StS_StD_LED => "Sz2_Button_LED_ST28_ST29",
              oHMI_status_StS_StD => "HMI_Pallets".Run_Status_left_ROW1[8],
              oHMI_status_StD_StS => "HMI_Pallets".Run_Status_right_ROW1[8],
              Stop_Drive_Button => "HMI_Pallets".Stop_Driver_Button1.%X28,
              Stop_Drive_HMI => "HMI_Pallets".Stop_Driver_HMI1.%X28);
END_REGION

REGION Network 71: ST27->ST28
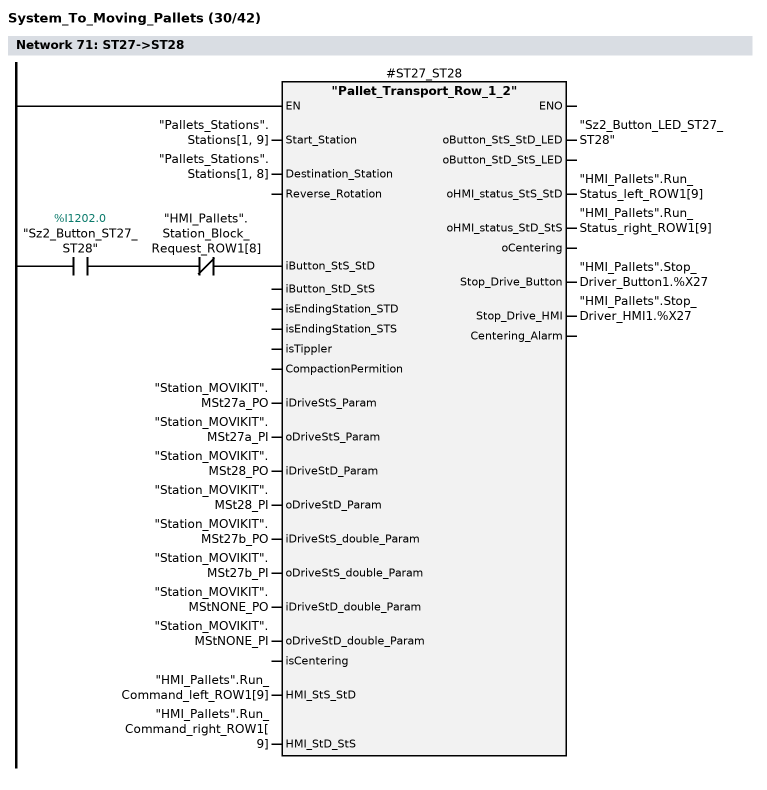
   RUNG wire#powerrail
      #ST27_ST28(iButton_StS_StD := wire#w1, Start_Station := "Pallets_Stations".Stations[1, 9], Destination_Station := "Pallets_Stations".Stations[1, 8], Reverse_Rotation :=, iButton_StD_StS :=, isEndingStation_STD :=, isEndingStation_STS :=, isTippler :=, CompactionPermition :=, iDriveStS_Param := "Station_MOVIKIT".MSt27a_PO, oDriveStS_Param := "Station_MOVIKIT".MSt27a_PI, iDriveStD_Param := "Station_MOVIKIT".MSt28_PO, oDriveStD_Param := "Station_MOVIKIT".MSt28_PI, iDriveStS_double_Param := "Station_MOVIKIT".MSt27b_PO, oDriveStS_double_Param := "Station_MOVIKIT".MSt27b_PI, iDriveStD_double_Param := "Station_MOVIKIT".MStNONE_PO, oDriveStD_double_Param := "Station_MOVIKIT".MStNONE_PI, isCentering :=, HMI_StS_StD := "HMI_Pallets".Run_Command_left_ROW1[9], HMI_StD_StS := "HMI_Pallets".Run_Command_right_ROW1[9], oButton_StS_StD_LED => "Sz2_Button_LED_ST27_ST28", oButton_StD_StS_LED =>, oHMI_status_StS_StD => "HMI_Pallets".Run_Status_left_ROW1[9], oHMI_status_StD_StS => "HMI_Pallets".Run_Status_right_ROW1[9], oCentering =>, Stop_Drive_Button => "HMI_Pallets".Stop_Driver_Button1.%X27, Stop_Drive_HMI => "HMI_Pallets".Stop_Driver_HMI1.%X27, Centering_Alarm =>)
   END_RUNG
   RUNG wire#powerrail
      Contact( "Sz2_Button_ST27_ST28" )
      I_Contact( "HMI_Pallets".Station_Block_Request_ROW1[8] )
   END_RUNG wire#w1
   // the same network as SCL:
   #ST27_ST28(Start_Station := "Pallets_Stations".Stations[1, 9],   // "Pallet_Transport_Row_1_2"
              Destination_Station := "Pallets_Stations".Stations[1, 8],
              iButton_StS_StD := "Sz2_Button_ST27_ST28" AND NOT "HMI_Pallets".Station_Block_Request_ROW1[8],
              iDriveStS_Param := "Station_MOVIKIT".MSt27a_PO,
              oDriveStS_Param := "Station_MOVIKIT".MSt27a_PI,
              iDriveStD_Param := "Station_MOVIKIT".MSt28_PO,
              oDriveStD_Param := "Station_MOVIKIT".MSt28_PI,
              iDriveStS_double_Param := "Station_MOVIKIT".MSt27b_PO,
              oDriveStS_double_Param := "Station_MOVIKIT".MSt27b_PI,
              iDriveStD_double_Param := "Station_MOVIKIT".MStNONE_PO,
              oDriveStD_double_Param := "Station_MOVIKIT".MStNONE_PI,
              HMI_StS_StD := "HMI_Pallets".Run_Command_left_ROW1[9],
              HMI_StD_StS := "HMI_Pallets".Run_Command_right_ROW1[9],
              oButton_StS_StD_LED => "Sz2_Button_LED_ST27_ST28",
              oHMI_status_StS_StD => "HMI_Pallets".Run_Status_left_ROW1[9],
              oHMI_status_StD_StS => "HMI_Pallets".Run_Status_right_ROW1[9],
              Stop_Drive_Button => "HMI_Pallets".Stop_Driver_Button1.%X27,
              Stop_Drive_HMI => "HMI_Pallets".Stop_Driver_HMI1.%X27);
END_REGION

REGION Network 72: ST26->ST27
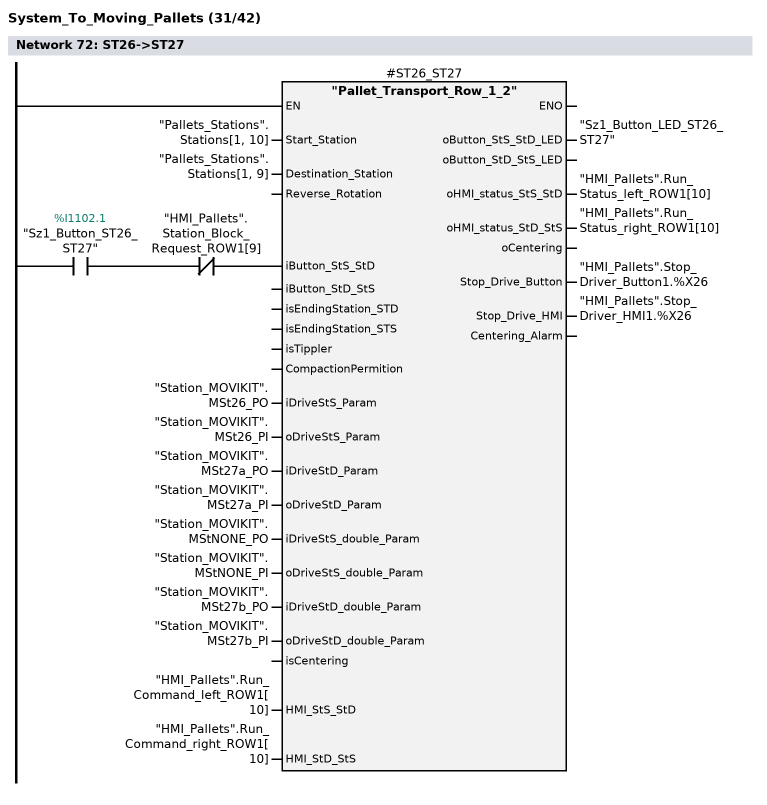
   RUNG wire#powerrail
      #ST26_ST27(iButton_StS_StD := wire#w1, Start_Station := "Pallets_Stations".Stations[1, 10], Destination_Station := "Pallets_Stations".Stations[1, 9], Reverse_Rotation :=, iButton_StD_StS :=, isEndingStation_STD :=, isEndingStation_STS :=, isTippler :=, CompactionPermition :=, iDriveStS_Param := "Station_MOVIKIT".MSt26_PO, oDriveStS_Param := "Station_MOVIKIT".MSt26_PI, iDriveStD_Param := "Station_MOVIKIT".MSt27a_PO, oDriveStD_Param := "Station_MOVIKIT".MSt27a_PI, iDriveStS_double_Param := "Station_MOVIKIT".MStNONE_PO, oDriveStS_double_Param := "Station_MOVIKIT".MStNONE_PI, iDriveStD_double_Param := "Station_MOVIKIT".MSt27b_PO, oDriveStD_double_Param := "Station_MOVIKIT".MSt27b_PI, isCentering :=, HMI_StS_StD := "HMI_Pallets".Run_Command_left_ROW1[10], HMI_StD_StS := "HMI_Pallets".Run_Command_right_ROW1[10], oButton_StS_StD_LED => "Sz1_Button_LED_ST26_ST27", oButton_StD_StS_LED =>, oHMI_status_StS_StD => "HMI_Pallets".Run_Status_left_ROW1[10], oHMI_status_StD_StS => "HMI_Pallets".Run_Status_right_ROW1[10], oCentering =>, Stop_Drive_Button => "HMI_Pallets".Stop_Driver_Button1.%X26, Stop_Drive_HMI => "HMI_Pallets".Stop_Driver_HMI1.%X26, Centering_Alarm =>)
   END_RUNG
   RUNG wire#powerrail
      Contact( "Sz1_Button_ST26_ST27" )
      I_Contact( "HMI_Pallets".Station_Block_Request_ROW1[9] )
   END_RUNG wire#w1
   // the same network as SCL:
   #ST26_ST27(Start_Station := "Pallets_Stations".Stations[1, 10],   // "Pallet_Transport_Row_1_2"
              Destination_Station := "Pallets_Stations".Stations[1, 9],
              iButton_StS_StD := "Sz1_Button_ST26_ST27" AND NOT "HMI_Pallets".Station_Block_Request_ROW1[9],
              iDriveStS_Param := "Station_MOVIKIT".MSt26_PO,
              oDriveStS_Param := "Station_MOVIKIT".MSt26_PI,
              iDriveStD_Param := "Station_MOVIKIT".MSt27a_PO,
              oDriveStD_Param := "Station_MOVIKIT".MSt27a_PI,
              iDriveStS_double_Param := "Station_MOVIKIT".MStNONE_PO,
              oDriveStS_double_Param := "Station_MOVIKIT".MStNONE_PI,
              iDriveStD_double_Param := "Station_MOVIKIT".MSt27b_PO,
              oDriveStD_double_Param := "Station_MOVIKIT".MSt27b_PI,
              HMI_StS_StD := "HMI_Pallets".Run_Command_left_ROW1[10],
              HMI_StD_StS := "HMI_Pallets".Run_Command_right_ROW1[10],
              oButton_StS_StD_LED => "Sz1_Button_LED_ST26_ST27",
              oHMI_status_StS_StD => "HMI_Pallets".Run_Status_left_ROW1[10],
              oHMI_status_StD_StS => "HMI_Pallets".Run_Status_right_ROW1[10],
              Stop_Drive_Button => "HMI_Pallets".Stop_Driver_Button1.%X26,
              Stop_Drive_HMI => "HMI_Pallets".Stop_Driver_HMI1.%X26);
END_REGION

REGION Network 73: ST25->ST26
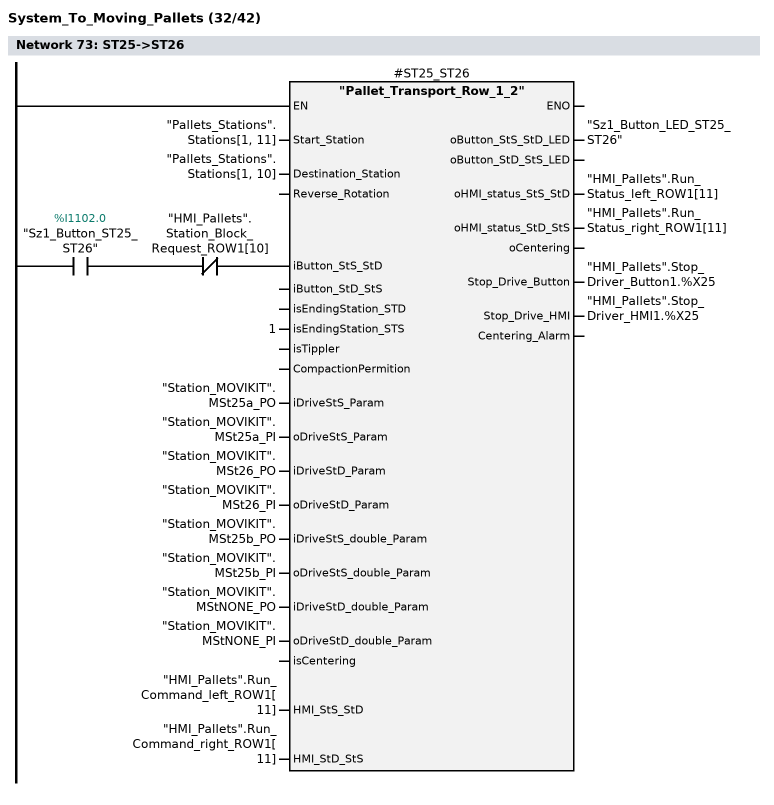
   RUNG wire#powerrail
      #ST25_ST26(iButton_StS_StD := wire#w1, Start_Station := "Pallets_Stations".Stations[1, 11], Destination_Station := "Pallets_Stations".Stations[1, 10], Reverse_Rotation :=, iButton_StD_StS :=, isEndingStation_STD :=, isEndingStation_STS := 1, isTippler :=, CompactionPermition :=, iDriveStS_Param := "Station_MOVIKIT".MSt25a_PO, oDriveStS_Param := "Station_MOVIKIT".MSt25a_PI, iDriveStD_Param := "Station_MOVIKIT".MSt26_PO, oDriveStD_Param := "Station_MOVIKIT".MSt26_PI, iDriveStS_double_Param := "Station_MOVIKIT".MSt25b_PO, oDriveStS_double_Param := "Station_MOVIKIT".MSt25b_PI, iDriveStD_double_Param := "Station_MOVIKIT".MStNONE_PO, oDriveStD_double_Param := "Station_MOVIKIT".MStNONE_PI, isCentering :=, HMI_StS_StD := "HMI_Pallets".Run_Command_left_ROW1[11], HMI_StD_StS := "HMI_Pallets".Run_Command_right_ROW1[11], oButton_StS_StD_LED => "Sz1_Button_LED_ST25_ST26", oButton_StD_StS_LED =>, oHMI_status_StS_StD => "HMI_Pallets".Run_Status_left_ROW1[11], oHMI_status_StD_StS => "HMI_Pallets".Run_Status_right_ROW1[11], oCentering =>, Stop_Drive_Button => "HMI_Pallets".Stop_Driver_Button1.%X25, Stop_Drive_HMI => "HMI_Pallets".Stop_Driver_HMI1.%X25, Centering_Alarm =>)
   END_RUNG
   RUNG wire#powerrail
      Contact( "Sz1_Button_ST25_ST26" )
      I_Contact( "HMI_Pallets".Station_Block_Request_ROW1[10] )
   END_RUNG wire#w1
   // the same network as SCL:
   #ST25_ST26(Start_Station := "Pallets_Stations".Stations[1, 11],   // "Pallet_Transport_Row_1_2"
              Destination_Station := "Pallets_Stations".Stations[1, 10],
              iButton_StS_StD := "Sz1_Button_ST25_ST26" AND NOT "HMI_Pallets".Station_Block_Request_ROW1[10],
              isEndingStation_STS := 1,
              iDriveStS_Param := "Station_MOVIKIT".MSt25a_PO,
              oDriveStS_Param := "Station_MOVIKIT".MSt25a_PI,
              iDriveStD_Param := "Station_MOVIKIT".MSt26_PO,
              oDriveStD_Param := "Station_MOVIKIT".MSt26_PI,
              iDriveStS_double_Param := "Station_MOVIKIT".MSt25b_PO,
              oDriveStS_double_Param := "Station_MOVIKIT".MSt25b_PI,
              iDriveStD_double_Param := "Station_MOVIKIT".MStNONE_PO,
              oDriveStD_double_Param := "Station_MOVIKIT".MStNONE_PI,
              HMI_StS_StD := "HMI_Pallets".Run_Command_left_ROW1[11],
              HMI_StD_StS := "HMI_Pallets".Run_Command_right_ROW1[11],
              oButton_StS_StD_LED => "Sz1_Button_LED_ST25_ST26",
              oHMI_status_StS_StD => "HMI_Pallets".Run_Status_left_ROW1[11],
              oHMI_status_StD_StS => "HMI_Pallets".Run_Status_right_ROW1[11],
              Stop_Drive_Button => "HMI_Pallets".Stop_Driver_Button1.%X25,
              Stop_Drive_HMI => "HMI_Pallets".Stop_Driver_HMI1.%X25);
END_REGION

REGION Network 74: ST36->ST38
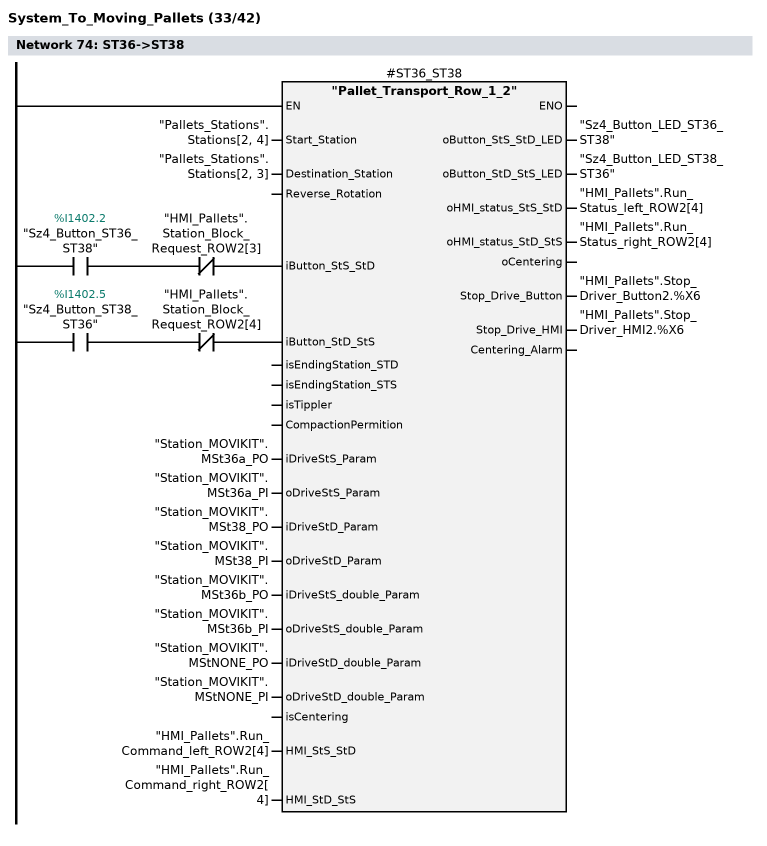
   RUNG wire#powerrail
      #ST36_ST38(iButton_StS_StD := wire#w1, iButton_StD_StS := wire#w2, Start_Station := "Pallets_Stations".Stations[2, 4], Destination_Station := "Pallets_Stations".Stations[2, 3], Reverse_Rotation :=, isEndingStation_STD :=, isEndingStation_STS :=, isTippler :=, CompactionPermition :=, iDriveStS_Param := "Station_MOVIKIT".MSt36a_PO, oDriveStS_Param := "Station_MOVIKIT".MSt36a_PI, iDriveStD_Param := "Station_MOVIKIT".MSt38_PO, oDriveStD_Param := "Station_MOVIKIT".MSt38_PI, iDriveStS_double_Param := "Station_MOVIKIT".MSt36b_PO, oDriveStS_double_Param := "Station_MOVIKIT".MSt36b_PI, iDriveStD_double_Param := "Station_MOVIKIT".MStNONE_PO, oDriveStD_double_Param := "Station_MOVIKIT".MStNONE_PI, isCentering :=, HMI_StS_StD := "HMI_Pallets".Run_Command_left_ROW2[4], HMI_StD_StS := "HMI_Pallets".Run_Command_right_ROW2[4], oButton_StS_StD_LED => "Sz4_Button_LED_ST36_ST38", oButton_StD_StS_LED => "Sz4_Button_LED_ST38_ST36", oHMI_status_StS_StD => "HMI_Pallets".Run_Status_left_ROW2[4], oHMI_status_StD_StS => "HMI_Pallets".Run_Status_right_ROW2[4], oCentering =>, Stop_Drive_Button => "HMI_Pallets".Stop_Driver_Button2.%X6, Stop_Drive_HMI => "HMI_Pallets".Stop_Driver_HMI2.%X6, Centering_Alarm =>)
   END_RUNG
   RUNG wire#powerrail
      Contact( "Sz4_Button_ST36_ST38" )
      I_Contact( "HMI_Pallets".Station_Block_Request_ROW2[3] )
   END_RUNG wire#w1
   RUNG wire#powerrail
      Contact( "Sz4_Button_ST38_ST36" )
      I_Contact( "HMI_Pallets".Station_Block_Request_ROW2[4] )
   END_RUNG wire#w2
   // the same network as SCL:
   #ST36_ST38(Start_Station := "Pallets_Stations".Stations[2, 4],   // "Pallet_Transport_Row_1_2"
              Destination_Station := "Pallets_Stations".Stations[2, 3],
              iButton_StS_StD := "Sz4_Button_ST36_ST38" AND NOT "HMI_Pallets".Station_Block_Request_ROW2[3],
              iButton_StD_StS := "Sz4_Button_ST38_ST36" AND NOT "HMI_Pallets".Station_Block_Request_ROW2[4],
              iDriveStS_Param := "Station_MOVIKIT".MSt36a_PO,
              oDriveStS_Param := "Station_MOVIKIT".MSt36a_PI,
              iDriveStD_Param := "Station_MOVIKIT".MSt38_PO,
              oDriveStD_Param := "Station_MOVIKIT".MSt38_PI,
              iDriveStS_double_Param := "Station_MOVIKIT".MSt36b_PO,
              oDriveStS_double_Param := "Station_MOVIKIT".MSt36b_PI,
              iDriveStD_double_Param := "Station_MOVIKIT".MStNONE_PO,
              oDriveStD_double_Param := "Station_MOVIKIT".MStNONE_PI,
              HMI_StS_StD := "HMI_Pallets".Run_Command_left_ROW2[4],
              HMI_StD_StS := "HMI_Pallets".Run_Command_right_ROW2[4],
              oButton_StS_StD_LED => "Sz4_Button_LED_ST36_ST38",
              oButton_StD_StS_LED => "Sz4_Button_LED_ST38_ST36",
              oHMI_status_StS_StD => "HMI_Pallets".Run_Status_left_ROW2[4],
              oHMI_status_StD_StS => "HMI_Pallets".Run_Status_right_ROW2[4],
              Stop_Drive_Button => "HMI_Pallets".Stop_Driver_Button2.%X6,
              Stop_Drive_HMI => "HMI_Pallets".Stop_Driver_HMI2.%X6);
END_REGION

REGION Network 75: ST37->ST36
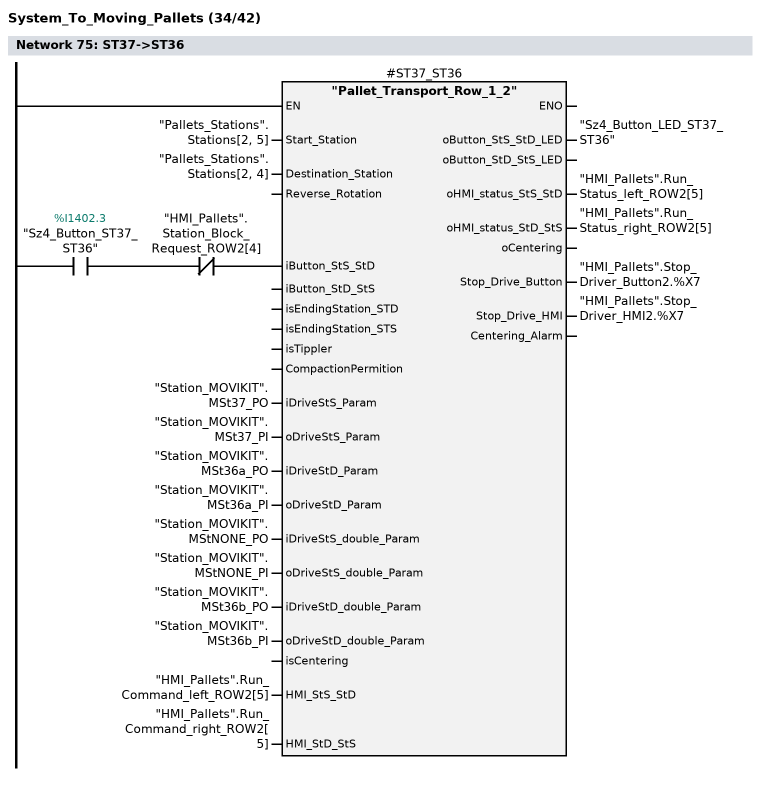
   RUNG wire#powerrail
      #ST37_ST36(iButton_StS_StD := wire#w1, Start_Station := "Pallets_Stations".Stations[2, 5], Destination_Station := "Pallets_Stations".Stations[2, 4], Reverse_Rotation :=, iButton_StD_StS :=, isEndingStation_STD :=, isEndingStation_STS :=, isTippler :=, CompactionPermition :=, iDriveStS_Param := "Station_MOVIKIT".MSt37_PO, oDriveStS_Param := "Station_MOVIKIT".MSt37_PI, iDriveStD_Param := "Station_MOVIKIT".MSt36a_PO, oDriveStD_Param := "Station_MOVIKIT".MSt36a_PI, iDriveStS_double_Param := "Station_MOVIKIT".MStNONE_PO, oDriveStS_double_Param := "Station_MOVIKIT".MStNONE_PI, iDriveStD_double_Param := "Station_MOVIKIT".MSt36b_PO, oDriveStD_double_Param := "Station_MOVIKIT".MSt36b_PI, isCentering :=, HMI_StS_StD := "HMI_Pallets".Run_Command_left_ROW2[5], HMI_StD_StS := "HMI_Pallets".Run_Command_right_ROW2[5], oButton_StS_StD_LED => "Sz4_Button_LED_ST37_ST36", oButton_StD_StS_LED =>, oHMI_status_StS_StD => "HMI_Pallets".Run_Status_left_ROW2[5], oHMI_status_StD_StS => "HMI_Pallets".Run_Status_right_ROW2[5], oCentering =>, Stop_Drive_Button => "HMI_Pallets".Stop_Driver_Button2.%X7, Stop_Drive_HMI => "HMI_Pallets".Stop_Driver_HMI2.%X7, Centering_Alarm =>)
   END_RUNG
   RUNG wire#powerrail
      Contact( "Sz4_Button_ST37_ST36" )
      I_Contact( "HMI_Pallets".Station_Block_Request_ROW2[4] )
   END_RUNG wire#w1
   // the same network as SCL:
   #ST37_ST36(Start_Station := "Pallets_Stations".Stations[2, 5],   // "Pallet_Transport_Row_1_2"
              Destination_Station := "Pallets_Stations".Stations[2, 4],
              iButton_StS_StD := "Sz4_Button_ST37_ST36" AND NOT "HMI_Pallets".Station_Block_Request_ROW2[4],
              iDriveStS_Param := "Station_MOVIKIT".MSt37_PO,
              oDriveStS_Param := "Station_MOVIKIT".MSt37_PI,
              iDriveStD_Param := "Station_MOVIKIT".MSt36a_PO,
              oDriveStD_Param := "Station_MOVIKIT".MSt36a_PI,
              iDriveStS_double_Param := "Station_MOVIKIT".MStNONE_PO,
              oDriveStS_double_Param := "Station_MOVIKIT".MStNONE_PI,
              iDriveStD_double_Param := "Station_MOVIKIT".MSt36b_PO,
              oDriveStD_double_Param := "Station_MOVIKIT".MSt36b_PI,
              HMI_StS_StD := "HMI_Pallets".Run_Command_left_ROW2[5],
              HMI_StD_StS := "HMI_Pallets".Run_Command_right_ROW2[5],
              oButton_StS_StD_LED => "Sz4_Button_LED_ST37_ST36",
              oHMI_status_StS_StD => "HMI_Pallets".Run_Status_left_ROW2[5],
              oHMI_status_StD_StS => "HMI_Pallets".Run_Status_right_ROW2[5],
              Stop_Drive_Button => "HMI_Pallets".Stop_Driver_Button2.%X7,
              Stop_Drive_HMI => "HMI_Pallets".Stop_Driver_HMI2.%X7);
END_REGION

REGION Network 76: ST18->ST37
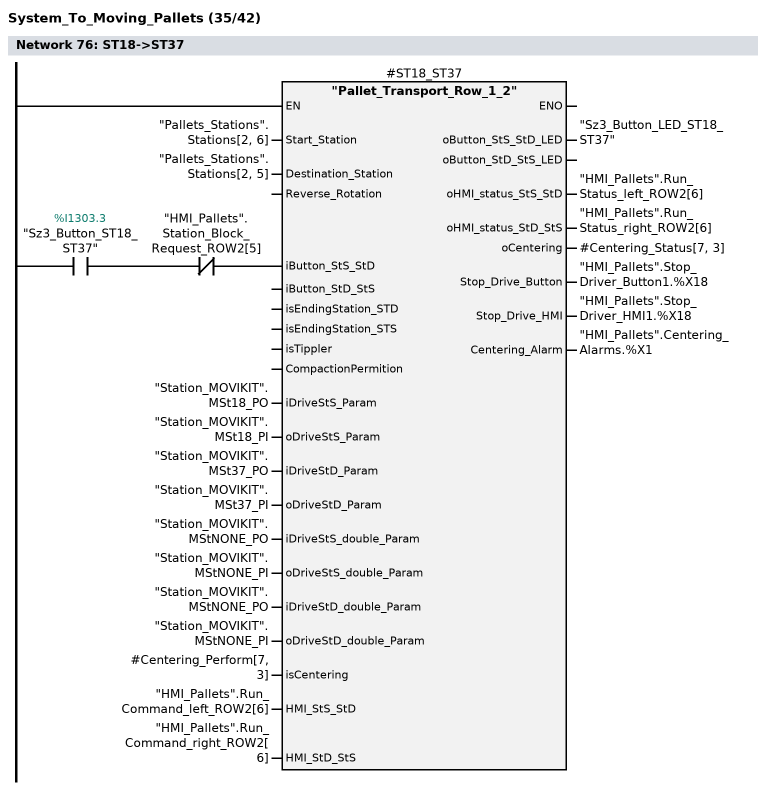
   RUNG wire#powerrail
      #ST18_ST37(iButton_StS_StD := wire#w1, Start_Station := "Pallets_Stations".Stations[2, 6], Destination_Station := "Pallets_Stations".Stations[2, 5], Reverse_Rotation :=, iButton_StD_StS :=, isEndingStation_STD :=, isEndingStation_STS :=, isTippler :=, CompactionPermition :=, iDriveStS_Param := "Station_MOVIKIT".MSt18_PO, oDriveStS_Param := "Station_MOVIKIT".MSt18_PI, iDriveStD_Param := "Station_MOVIKIT".MSt37_PO, oDriveStD_Param := "Station_MOVIKIT".MSt37_PI, iDriveStS_double_Param := "Station_MOVIKIT".MStNONE_PO, oDriveStS_double_Param := "Station_MOVIKIT".MStNONE_PI, iDriveStD_double_Param := "Station_MOVIKIT".MStNONE_PO, oDriveStD_double_Param := "Station_MOVIKIT".MStNONE_PI, isCentering := #Centering_Perform[7, 3], HMI_StS_StD := "HMI_Pallets".Run_Command_left_ROW2[6], HMI_StD_StS := "HMI_Pallets".Run_Command_right_ROW2[6], oButton_StS_StD_LED => "Sz3_Button_LED_ST18_ST37", oButton_StD_StS_LED =>, oHMI_status_StS_StD => "HMI_Pallets".Run_Status_left_ROW2[6], oHMI_status_StD_StS => "HMI_Pallets".Run_Status_right_ROW2[6], oCentering => #Centering_Status[7, 3], Stop_Drive_Button => "HMI_Pallets".Stop_Driver_Button1.%X18, Stop_Drive_HMI => "HMI_Pallets".Stop_Driver_HMI1.%X18, Centering_Alarm => "HMI_Pallets".Centering_Alarms.%X1)
   END_RUNG
   RUNG wire#powerrail
      Contact( "Sz3_Button_ST18_ST37" )
      I_Contact( "HMI_Pallets".Station_Block_Request_ROW2[5] )
   END_RUNG wire#w1
   // the same network as SCL:
   #ST18_ST37(Start_Station := "Pallets_Stations".Stations[2, 6],   // "Pallet_Transport_Row_1_2"
              Destination_Station := "Pallets_Stations".Stations[2, 5],
              iButton_StS_StD := "Sz3_Button_ST18_ST37" AND NOT "HMI_Pallets".Station_Block_Request_ROW2[5],
              iDriveStS_Param := "Station_MOVIKIT".MSt18_PO,
              oDriveStS_Param := "Station_MOVIKIT".MSt18_PI,
              iDriveStD_Param := "Station_MOVIKIT".MSt37_PO,
              oDriveStD_Param := "Station_MOVIKIT".MSt37_PI,
              iDriveStS_double_Param := "Station_MOVIKIT".MStNONE_PO,
              oDriveStS_double_Param := "Station_MOVIKIT".MStNONE_PI,
              iDriveStD_double_Param := "Station_MOVIKIT".MStNONE_PO,
              oDriveStD_double_Param := "Station_MOVIKIT".MStNONE_PI,
              isCentering := #Centering_Perform[7, 3],
              HMI_StS_StD := "HMI_Pallets".Run_Command_left_ROW2[6],
              HMI_StD_StS := "HMI_Pallets".Run_Command_right_ROW2[6],
              oButton_StS_StD_LED => "Sz3_Button_LED_ST18_ST37",
              oHMI_status_StS_StD => "HMI_Pallets".Run_Status_left_ROW2[6],
              oHMI_status_StD_StS => "HMI_Pallets".Run_Status_right_ROW2[6],
              oCentering => #Centering_Status[7, 3],
              Stop_Drive_Button => "HMI_Pallets".Stop_Driver_Button1.%X18,
              Stop_Drive_HMI => "HMI_Pallets".Stop_Driver_HMI1.%X18,
              Centering_Alarm => "HMI_Pallets".Centering_Alarms.%X1);
END_REGION

REGION Network 77: ST19->ST18
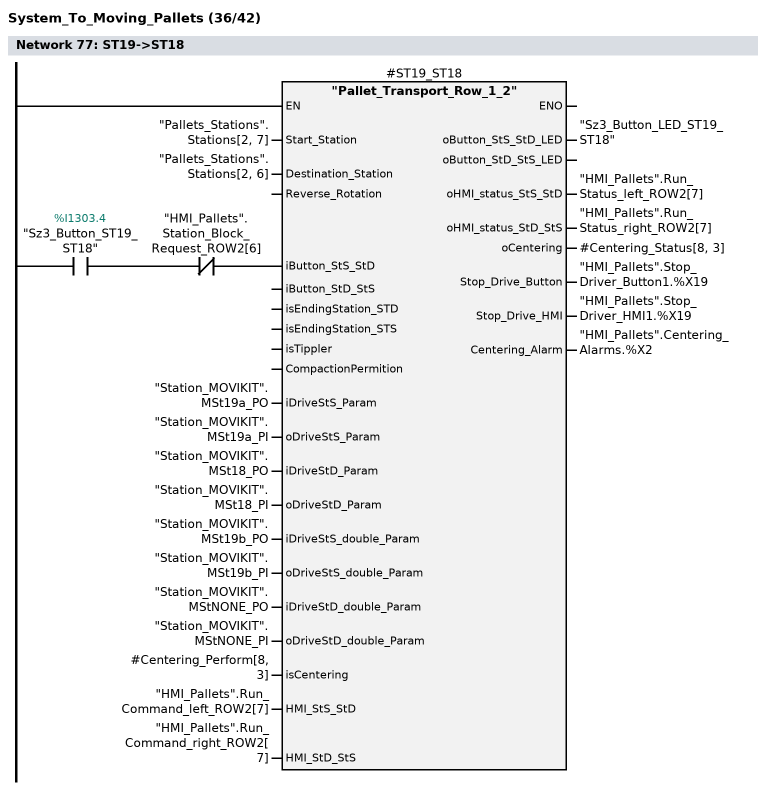
   RUNG wire#powerrail
      #ST19_ST18(iButton_StS_StD := wire#w1, Start_Station := "Pallets_Stations".Stations[2, 7], Destination_Station := "Pallets_Stations".Stations[2, 6], Reverse_Rotation :=, iButton_StD_StS :=, isEndingStation_STD :=, isEndingStation_STS :=, isTippler :=, CompactionPermition :=, iDriveStS_Param := "Station_MOVIKIT".MSt19a_PO, oDriveStS_Param := "Station_MOVIKIT".MSt19a_PI, iDriveStD_Param := "Station_MOVIKIT".MSt18_PO, oDriveStD_Param := "Station_MOVIKIT".MSt18_PI, iDriveStS_double_Param := "Station_MOVIKIT".MSt19b_PO, oDriveStS_double_Param := "Station_MOVIKIT".MSt19b_PI, iDriveStD_double_Param := "Station_MOVIKIT".MStNONE_PO, oDriveStD_double_Param := "Station_MOVIKIT".MStNONE_PI, isCentering := #Centering_Perform[8, 3], HMI_StS_StD := "HMI_Pallets".Run_Command_left_ROW2[7], HMI_StD_StS := "HMI_Pallets".Run_Command_right_ROW2[7], oButton_StS_StD_LED => "Sz3_Button_LED_ST19_ST18", oButton_StD_StS_LED =>, oHMI_status_StS_StD => "HMI_Pallets".Run_Status_left_ROW2[7], oHMI_status_StD_StS => "HMI_Pallets".Run_Status_right_ROW2[7], oCentering => #Centering_Status[8, 3], Stop_Drive_Button => "HMI_Pallets".Stop_Driver_Button1.%X19, Stop_Drive_HMI => "HMI_Pallets".Stop_Driver_HMI1.%X19, Centering_Alarm => "HMI_Pallets".Centering_Alarms.%X2)
   END_RUNG
   RUNG wire#powerrail
      Contact( "Sz3_Button_ST19_ST18" )
      I_Contact( "HMI_Pallets".Station_Block_Request_ROW2[6] )
   END_RUNG wire#w1
   // the same network as SCL:
   #ST19_ST18(Start_Station := "Pallets_Stations".Stations[2, 7],   // "Pallet_Transport_Row_1_2"
              Destination_Station := "Pallets_Stations".Stations[2, 6],
              iButton_StS_StD := "Sz3_Button_ST19_ST18" AND NOT "HMI_Pallets".Station_Block_Request_ROW2[6],
              iDriveStS_Param := "Station_MOVIKIT".MSt19a_PO,
              oDriveStS_Param := "Station_MOVIKIT".MSt19a_PI,
              iDriveStD_Param := "Station_MOVIKIT".MSt18_PO,
              oDriveStD_Param := "Station_MOVIKIT".MSt18_PI,
              iDriveStS_double_Param := "Station_MOVIKIT".MSt19b_PO,
              oDriveStS_double_Param := "Station_MOVIKIT".MSt19b_PI,
              iDriveStD_double_Param := "Station_MOVIKIT".MStNONE_PO,
              oDriveStD_double_Param := "Station_MOVIKIT".MStNONE_PI,
              isCentering := #Centering_Perform[8, 3],
              HMI_StS_StD := "HMI_Pallets".Run_Command_left_ROW2[7],
              HMI_StD_StS := "HMI_Pallets".Run_Command_right_ROW2[7],
              oButton_StS_StD_LED => "Sz3_Button_LED_ST19_ST18",
              oHMI_status_StS_StD => "HMI_Pallets".Run_Status_left_ROW2[7],
              oHMI_status_StD_StS => "HMI_Pallets".Run_Status_right_ROW2[7],
              oCentering => #Centering_Status[8, 3],
              Stop_Drive_Button => "HMI_Pallets".Stop_Driver_Button1.%X19,
              Stop_Drive_HMI => "HMI_Pallets".Stop_Driver_HMI1.%X19,
              Centering_Alarm => "HMI_Pallets".Centering_Alarms.%X2);
END_REGION

REGION Network 78: ST20->ST19
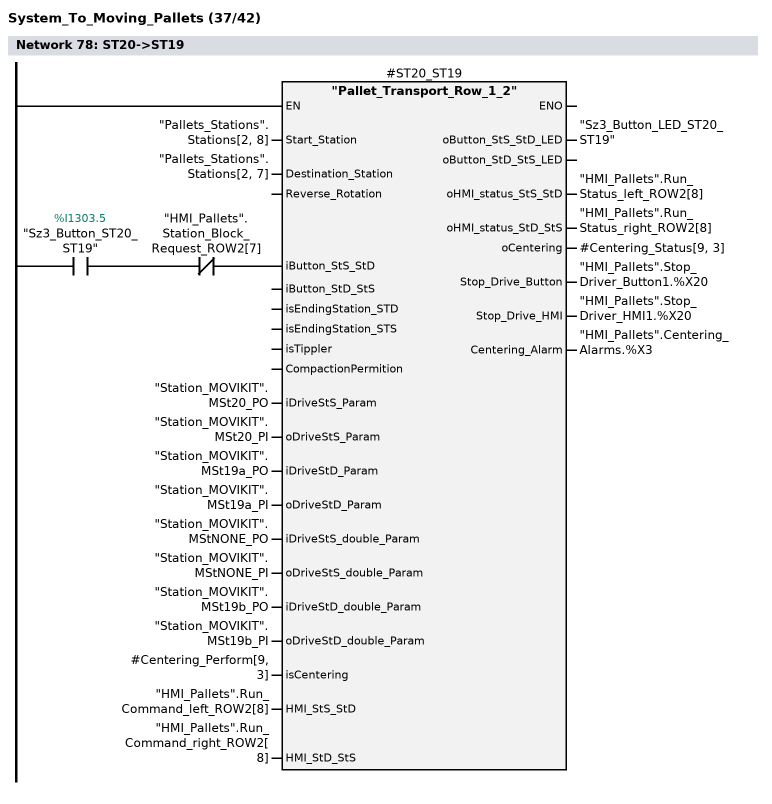
   RUNG wire#powerrail
      #ST20_ST19(iButton_StS_StD := wire#w1, Start_Station := "Pallets_Stations".Stations[2, 8], Destination_Station := "Pallets_Stations".Stations[2, 7], Reverse_Rotation :=, iButton_StD_StS :=, isEndingStation_STD :=, isEndingStation_STS :=, isTippler :=, CompactionPermition :=, iDriveStS_Param := "Station_MOVIKIT".MSt20_PO, oDriveStS_Param := "Station_MOVIKIT".MSt20_PI, iDriveStD_Param := "Station_MOVIKIT".MSt19a_PO, oDriveStD_Param := "Station_MOVIKIT".MSt19a_PI, iDriveStS_double_Param := "Station_MOVIKIT".MStNONE_PO, oDriveStS_double_Param := "Station_MOVIKIT".MStNONE_PI, iDriveStD_double_Param := "Station_MOVIKIT".MSt19b_PO, oDriveStD_double_Param := "Station_MOVIKIT".MSt19b_PI, isCentering := #Centering_Perform[9, 3], HMI_StS_StD := "HMI_Pallets".Run_Command_left_ROW2[8], HMI_StD_StS := "HMI_Pallets".Run_Command_right_ROW2[8], oButton_StS_StD_LED => "Sz3_Button_LED_ST20_ST19", oButton_StD_StS_LED =>, oHMI_status_StS_StD => "HMI_Pallets".Run_Status_left_ROW2[8], oHMI_status_StD_StS => "HMI_Pallets".Run_Status_right_ROW2[8], oCentering => #Centering_Status[9, 3], Stop_Drive_Button => "HMI_Pallets".Stop_Driver_Button1.%X20, Stop_Drive_HMI => "HMI_Pallets".Stop_Driver_HMI1.%X20, Centering_Alarm => "HMI_Pallets".Centering_Alarms.%X3)
   END_RUNG
   RUNG wire#powerrail
      Contact( "Sz3_Button_ST20_ST19" )
      I_Contact( "HMI_Pallets".Station_Block_Request_ROW2[7] )
   END_RUNG wire#w1
   // the same network as SCL:
   #ST20_ST19(Start_Station := "Pallets_Stations".Stations[2, 8],   // "Pallet_Transport_Row_1_2"
              Destination_Station := "Pallets_Stations".Stations[2, 7],
              iButton_StS_StD := "Sz3_Button_ST20_ST19" AND NOT "HMI_Pallets".Station_Block_Request_ROW2[7],
              iDriveStS_Param := "Station_MOVIKIT".MSt20_PO,
              oDriveStS_Param := "Station_MOVIKIT".MSt20_PI,
              iDriveStD_Param := "Station_MOVIKIT".MSt19a_PO,
              oDriveStD_Param := "Station_MOVIKIT".MSt19a_PI,
              iDriveStS_double_Param := "Station_MOVIKIT".MStNONE_PO,
              oDriveStS_double_Param := "Station_MOVIKIT".MStNONE_PI,
              iDriveStD_double_Param := "Station_MOVIKIT".MSt19b_PO,
              oDriveStD_double_Param := "Station_MOVIKIT".MSt19b_PI,
              isCentering := #Centering_Perform[9, 3],
              HMI_StS_StD := "HMI_Pallets".Run_Command_left_ROW2[8],
              HMI_StD_StS := "HMI_Pallets".Run_Command_right_ROW2[8],
              oButton_StS_StD_LED => "Sz3_Button_LED_ST20_ST19",
              oHMI_status_StS_StD => "HMI_Pallets".Run_Status_left_ROW2[8],
              oHMI_status_StD_StS => "HMI_Pallets".Run_Status_right_ROW2[8],
              oCentering => #Centering_Status[9, 3],
              Stop_Drive_Button => "HMI_Pallets".Stop_Driver_Button1.%X20,
              Stop_Drive_HMI => "HMI_Pallets".Stop_Driver_HMI1.%X20,
              Centering_Alarm => "HMI_Pallets".Centering_Alarms.%X3);
END_REGION

REGION Network 79: ST21->ST20
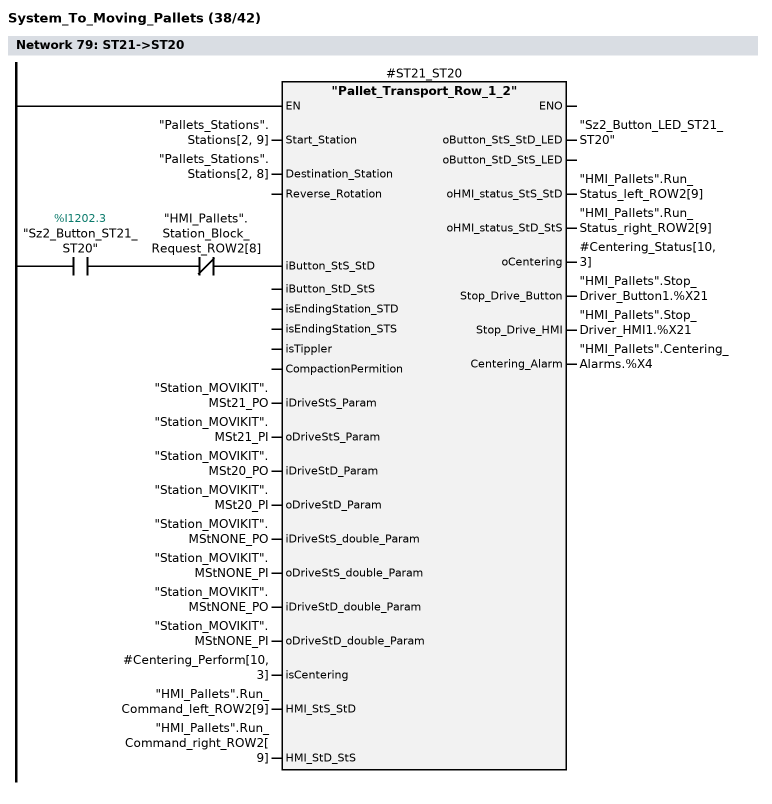
   RUNG wire#powerrail
      #ST21_ST20(iButton_StS_StD := wire#w1, Start_Station := "Pallets_Stations".Stations[2, 9], Destination_Station := "Pallets_Stations".Stations[2, 8], Reverse_Rotation :=, iButton_StD_StS :=, isEndingStation_STD :=, isEndingStation_STS :=, isTippler :=, CompactionPermition :=, iDriveStS_Param := "Station_MOVIKIT".MSt21_PO, oDriveStS_Param := "Station_MOVIKIT".MSt21_PI, iDriveStD_Param := "Station_MOVIKIT".MSt20_PO, oDriveStD_Param := "Station_MOVIKIT".MSt20_PI, iDriveStS_double_Param := "Station_MOVIKIT".MStNONE_PO, oDriveStS_double_Param := "Station_MOVIKIT".MStNONE_PI, iDriveStD_double_Param := "Station_MOVIKIT".MStNONE_PO, oDriveStD_double_Param := "Station_MOVIKIT".MStNONE_PI, isCentering := #Centering_Perform[10, 3], HMI_StS_StD := "HMI_Pallets".Run_Command_left_ROW2[9], HMI_StD_StS := "HMI_Pallets".Run_Command_right_ROW2[9], oButton_StS_StD_LED => "Sz2_Button_LED_ST21_ST20", oButton_StD_StS_LED =>, oHMI_status_StS_StD => "HMI_Pallets".Run_Status_left_ROW2[9], oHMI_status_StD_StS => "HMI_Pallets".Run_Status_right_ROW2[9], oCentering => #Centering_Status[10, 3], Stop_Drive_Button => "HMI_Pallets".Stop_Driver_Button1.%X21, Stop_Drive_HMI => "HMI_Pallets".Stop_Driver_HMI1.%X21, Centering_Alarm => "HMI_Pallets".Centering_Alarms.%X4)
   END_RUNG
   RUNG wire#powerrail
      Contact( "Sz2_Button_ST21_ST20" )
      I_Contact( "HMI_Pallets".Station_Block_Request_ROW2[8] )
   END_RUNG wire#w1
   // the same network as SCL:
   #ST21_ST20(Start_Station := "Pallets_Stations".Stations[2, 9],   // "Pallet_Transport_Row_1_2"
              Destination_Station := "Pallets_Stations".Stations[2, 8],
              iButton_StS_StD := "Sz2_Button_ST21_ST20" AND NOT "HMI_Pallets".Station_Block_Request_ROW2[8],
              iDriveStS_Param := "Station_MOVIKIT".MSt21_PO,
              oDriveStS_Param := "Station_MOVIKIT".MSt21_PI,
              iDriveStD_Param := "Station_MOVIKIT".MSt20_PO,
              oDriveStD_Param := "Station_MOVIKIT".MSt20_PI,
              iDriveStS_double_Param := "Station_MOVIKIT".MStNONE_PO,
              oDriveStS_double_Param := "Station_MOVIKIT".MStNONE_PI,
              iDriveStD_double_Param := "Station_MOVIKIT".MStNONE_PO,
              oDriveStD_double_Param := "Station_MOVIKIT".MStNONE_PI,
              isCentering := #Centering_Perform[10, 3],
              HMI_StS_StD := "HMI_Pallets".Run_Command_left_ROW2[9],
              HMI_StD_StS := "HMI_Pallets".Run_Command_right_ROW2[9],
              oButton_StS_StD_LED => "Sz2_Button_LED_ST21_ST20",
              oHMI_status_StS_StD => "HMI_Pallets".Run_Status_left_ROW2[9],
              oHMI_status_StD_StS => "HMI_Pallets".Run_Status_right_ROW2[9],
              oCentering => #Centering_Status[10, 3],
              Stop_Drive_Button => "HMI_Pallets".Stop_Driver_Button1.%X21,
              Stop_Drive_HMI => "HMI_Pallets".Stop_Driver_HMI1.%X21,
              Centering_Alarm => "HMI_Pallets".Centering_Alarms.%X4);
END_REGION

REGION Network 80: ST22->ST21
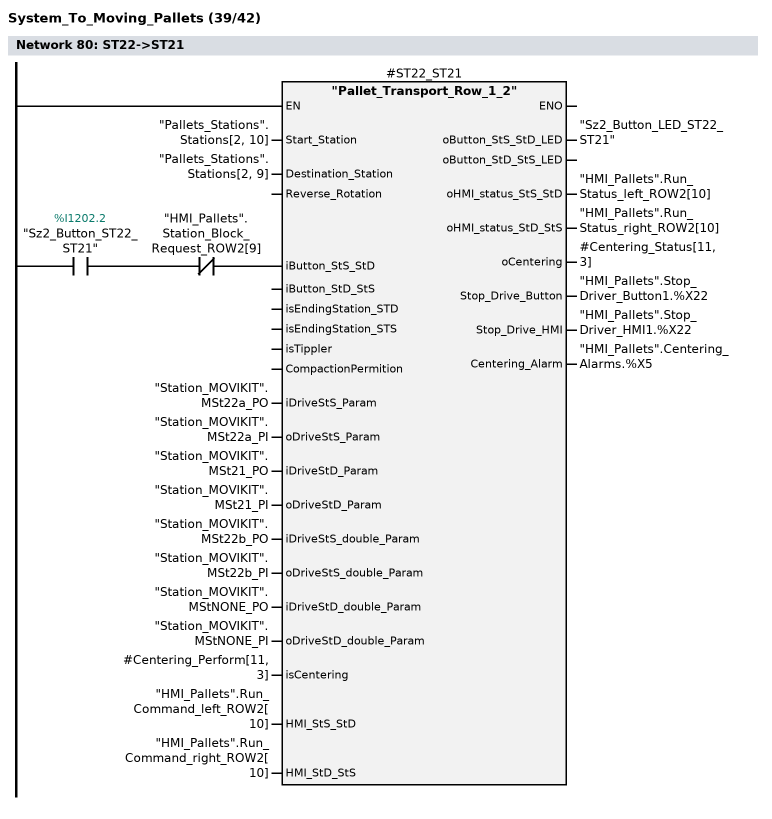
   RUNG wire#powerrail
      #ST22_ST21(iButton_StS_StD := wire#w1, Start_Station := "Pallets_Stations".Stations[2, 10], Destination_Station := "Pallets_Stations".Stations[2, 9], Reverse_Rotation :=, iButton_StD_StS :=, isEndingStation_STD :=, isEndingStation_STS :=, isTippler :=, CompactionPermition :=, iDriveStS_Param := "Station_MOVIKIT".MSt22a_PO, oDriveStS_Param := "Station_MOVIKIT".MSt22a_PI, iDriveStD_Param := "Station_MOVIKIT".MSt21_PO, oDriveStD_Param := "Station_MOVIKIT".MSt21_PI, iDriveStS_double_Param := "Station_MOVIKIT".MSt22b_PO, oDriveStS_double_Param := "Station_MOVIKIT".MSt22b_PI, iDriveStD_double_Param := "Station_MOVIKIT".MStNONE_PO, oDriveStD_double_Param := "Station_MOVIKIT".MStNONE_PI, isCentering := #Centering_Perform[11, 3], HMI_StS_StD := "HMI_Pallets".Run_Command_left_ROW2[10], HMI_StD_StS := "HMI_Pallets".Run_Command_right_ROW2[10], oButton_StS_StD_LED => "Sz2_Button_LED_ST22_ST21", oButton_StD_StS_LED =>, oHMI_status_StS_StD => "HMI_Pallets".Run_Status_left_ROW2[10], oHMI_status_StD_StS => "HMI_Pallets".Run_Status_right_ROW2[10], oCentering => #Centering_Status[11, 3], Stop_Drive_Button => "HMI_Pallets".Stop_Driver_Button1.%X22, Stop_Drive_HMI => "HMI_Pallets".Stop_Driver_HMI1.%X22, Centering_Alarm => "HMI_Pallets".Centering_Alarms.%X5)
   END_RUNG
   RUNG wire#powerrail
      Contact( "Sz2_Button_ST22_ST21" )
      I_Contact( "HMI_Pallets".Station_Block_Request_ROW2[9] )
   END_RUNG wire#w1
   // the same network as SCL:
   #ST22_ST21(Start_Station := "Pallets_Stations".Stations[2, 10],   // "Pallet_Transport_Row_1_2"
              Destination_Station := "Pallets_Stations".Stations[2, 9],
              iButton_StS_StD := "Sz2_Button_ST22_ST21" AND NOT "HMI_Pallets".Station_Block_Request_ROW2[9],
              iDriveStS_Param := "Station_MOVIKIT".MSt22a_PO,
              oDriveStS_Param := "Station_MOVIKIT".MSt22a_PI,
              iDriveStD_Param := "Station_MOVIKIT".MSt21_PO,
              oDriveStD_Param := "Station_MOVIKIT".MSt21_PI,
              iDriveStS_double_Param := "Station_MOVIKIT".MSt22b_PO,
              oDriveStS_double_Param := "Station_MOVIKIT".MSt22b_PI,
              iDriveStD_double_Param := "Station_MOVIKIT".MStNONE_PO,
              oDriveStD_double_Param := "Station_MOVIKIT".MStNONE_PI,
              isCentering := #Centering_Perform[11, 3],
              HMI_StS_StD := "HMI_Pallets".Run_Command_left_ROW2[10],
              HMI_StD_StS := "HMI_Pallets".Run_Command_right_ROW2[10],
              oButton_StS_StD_LED => "Sz2_Button_LED_ST22_ST21",
              oHMI_status_StS_StD => "HMI_Pallets".Run_Status_left_ROW2[10],
              oHMI_status_StD_StS => "HMI_Pallets".Run_Status_right_ROW2[10],
              oCentering => #Centering_Status[11, 3],
              Stop_Drive_Button => "HMI_Pallets".Stop_Driver_Button1.%X22,
              Stop_Drive_HMI => "HMI_Pallets".Stop_Driver_HMI1.%X22,
              Centering_Alarm => "HMI_Pallets".Centering_Alarms.%X5);
END_REGION

REGION Network 81: ST23->ST22
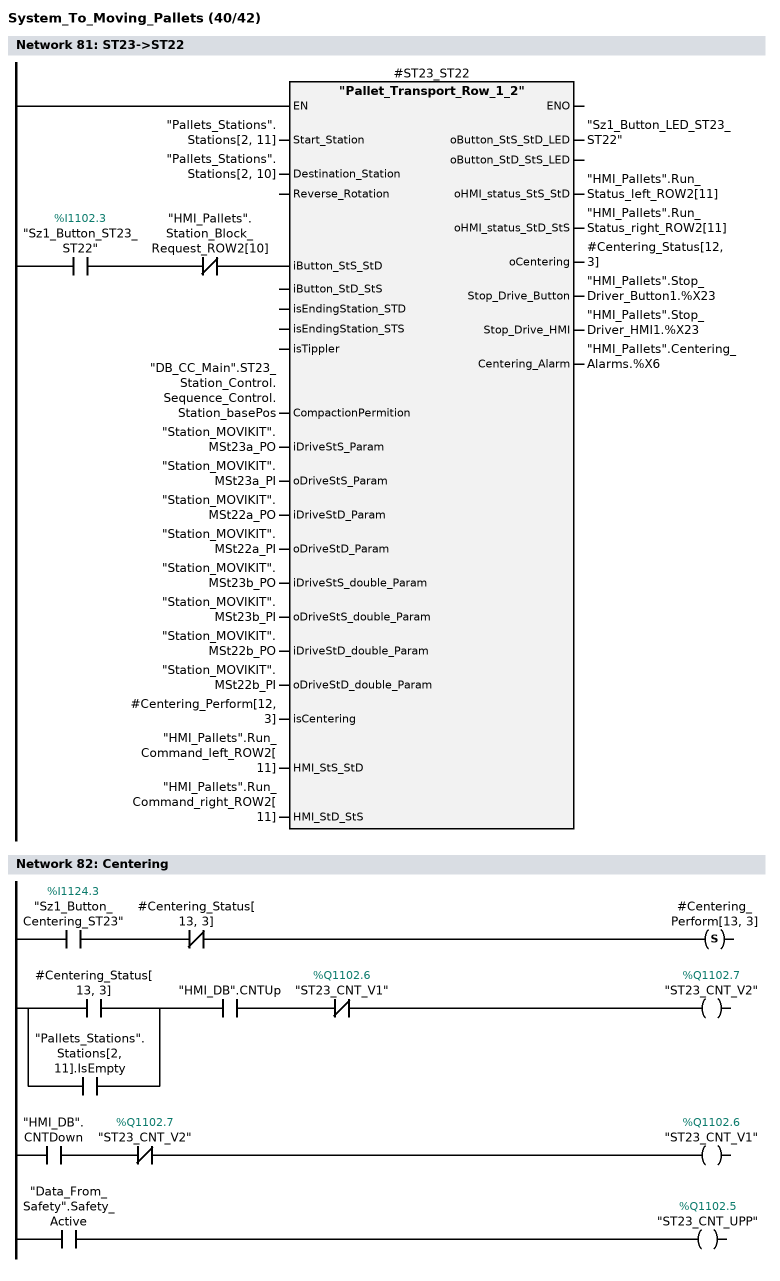
   RUNG wire#powerrail
      #ST23_ST22(iButton_StS_StD := wire#w1, Start_Station := "Pallets_Stations".Stations[2, 11], Destination_Station := "Pallets_Stations".Stations[2, 10], Reverse_Rotation :=, iButton_StD_StS :=, isEndingStation_STD :=, isEndingStation_STS :=, isTippler :=, CompactionPermition := "DB_CC_Main".ST23_Station_Control.Sequence_Control.Station_basePos, iDriveStS_Param := "Station_MOVIKIT".MSt23a_PO, oDriveStS_Param := "Station_MOVIKIT".MSt23a_PI, iDriveStD_Param := "Station_MOVIKIT".MSt22a_PO, oDriveStD_Param := "Station_MOVIKIT".MSt22a_PI, iDriveStS_double_Param := "Station_MOVIKIT".MSt23b_PO, oDriveStS_double_Param := "Station_MOVIKIT".MSt23b_PI, iDriveStD_double_Param := "Station_MOVIKIT".MSt22b_PO, oDriveStD_double_Param := "Station_MOVIKIT".MSt22b_PI, isCentering := #Centering_Perform[12, 3], HMI_StS_StD := "HMI_Pallets".Run_Command_left_ROW2[11], HMI_StD_StS := "HMI_Pallets".Run_Command_right_ROW2[11], oButton_StS_StD_LED => "Sz1_Button_LED_ST23_ST22", oButton_StD_StS_LED =>, oHMI_status_StS_StD => "HMI_Pallets".Run_Status_left_ROW2[11], oHMI_status_StD_StS => "HMI_Pallets".Run_Status_right_ROW2[11], oCentering => #Centering_Status[12, 3], Stop_Drive_Button => "HMI_Pallets".Stop_Driver_Button1.%X23, Stop_Drive_HMI => "HMI_Pallets".Stop_Driver_HMI1.%X23, Centering_Alarm => "HMI_Pallets".Centering_Alarms.%X6)
   END_RUNG
   RUNG wire#powerrail
      Contact( "Sz1_Button_ST23_ST22" )
      I_Contact( "HMI_Pallets".Station_Block_Request_ROW2[10] )
   END_RUNG wire#w1
   // the same network as SCL:
   #ST23_ST22(Start_Station := "Pallets_Stations".Stations[2, 11],   // "Pallet_Transport_Row_1_2"
              Destination_Station := "Pallets_Stations".Stations[2, 10],
              iButton_StS_StD := "Sz1_Button_ST23_ST22" AND NOT "HMI_Pallets".Station_Block_Request_ROW2[10],
              CompactionPermition := "DB_CC_Main".ST23_Station_Control.Sequence_Control.Station_basePos,
              iDriveStS_Param := "Station_MOVIKIT".MSt23a_PO,
              oDriveStS_Param := "Station_MOVIKIT".MSt23a_PI,
              iDriveStD_Param := "Station_MOVIKIT".MSt22a_PO,
              oDriveStD_Param := "Station_MOVIKIT".MSt22a_PI,
              iDriveStS_double_Param := "Station_MOVIKIT".MSt23b_PO,
              oDriveStS_double_Param := "Station_MOVIKIT".MSt23b_PI,
              iDriveStD_double_Param := "Station_MOVIKIT".MSt22b_PO,
              oDriveStD_double_Param := "Station_MOVIKIT".MSt22b_PI,
              isCentering := #Centering_Perform[12, 3],
              HMI_StS_StD := "HMI_Pallets".Run_Command_left_ROW2[11],
              HMI_StD_StS := "HMI_Pallets".Run_Command_right_ROW2[11],
              oButton_StS_StD_LED => "Sz1_Button_LED_ST23_ST22",
              oHMI_status_StS_StD => "HMI_Pallets".Run_Status_left_ROW2[11],
              oHMI_status_StD_StS => "HMI_Pallets".Run_Status_right_ROW2[11],
              oCentering => #Centering_Status[12, 3],
              Stop_Drive_Button => "HMI_Pallets".Stop_Driver_Button1.%X23,
              Stop_Drive_HMI => "HMI_Pallets".Stop_Driver_HMI1.%X23,
              Centering_Alarm => "HMI_Pallets".Centering_Alarms.%X6);
END_REGION

REGION Network 82: Centering
   RUNG wire#powerrail
      Contact( "Sz1_Button_Centering_ST23" )
      I_Contact( #Centering_Status[13, 3] )
      S_Coil( #Centering_Perform[13, 3] )
   END_RUNG
   RUNG wire#powerrail
      Contact( #Centering_Status[13, 3] )
      wire#w1
      Contact( "HMI_DB".CNTUp )
      I_Contact( "ST23_CNT_V1" )
      Coil( "ST23_CNT_V2" )
   END_RUNG
   RUNG wire#powerrail
      Contact( "Pallets_Stations".Stations[2, 11].IsEmpty )
   END_RUNG wire#w1
   RUNG wire#powerrail
      Contact( "HMI_DB".CNTDown )
      I_Contact( "ST23_CNT_V2" )
      Coil( "ST23_CNT_V1" )
   END_RUNG
   RUNG wire#powerrail
      Contact( "Data_From_Safety".Safety_Active )
      Coil( "ST23_CNT_UPP" )
   END_RUNG
   // the same network as SCL:
   IF "Sz1_Button_Centering_ST23" AND NOT #Centering_Status[13, 3] THEN
       #Centering_Perform[13, 3] := TRUE;
   END_IF;
   "ST23_CNT_V2" := (#Centering_Status[13, 3] OR "Pallets_Stations".Stations[2, 11].IsEmpty) AND "HMI_DB".CNTUp AND NOT "ST23_CNT_V1";
   "ST23_CNT_V1" := "HMI_DB".CNTDown AND NOT "ST23_CNT_V2";
   "ST23_CNT_UPP" := "Data_From_Safety".Safety_Active;
END_REGION

REGION Network 83: ST24->ST23
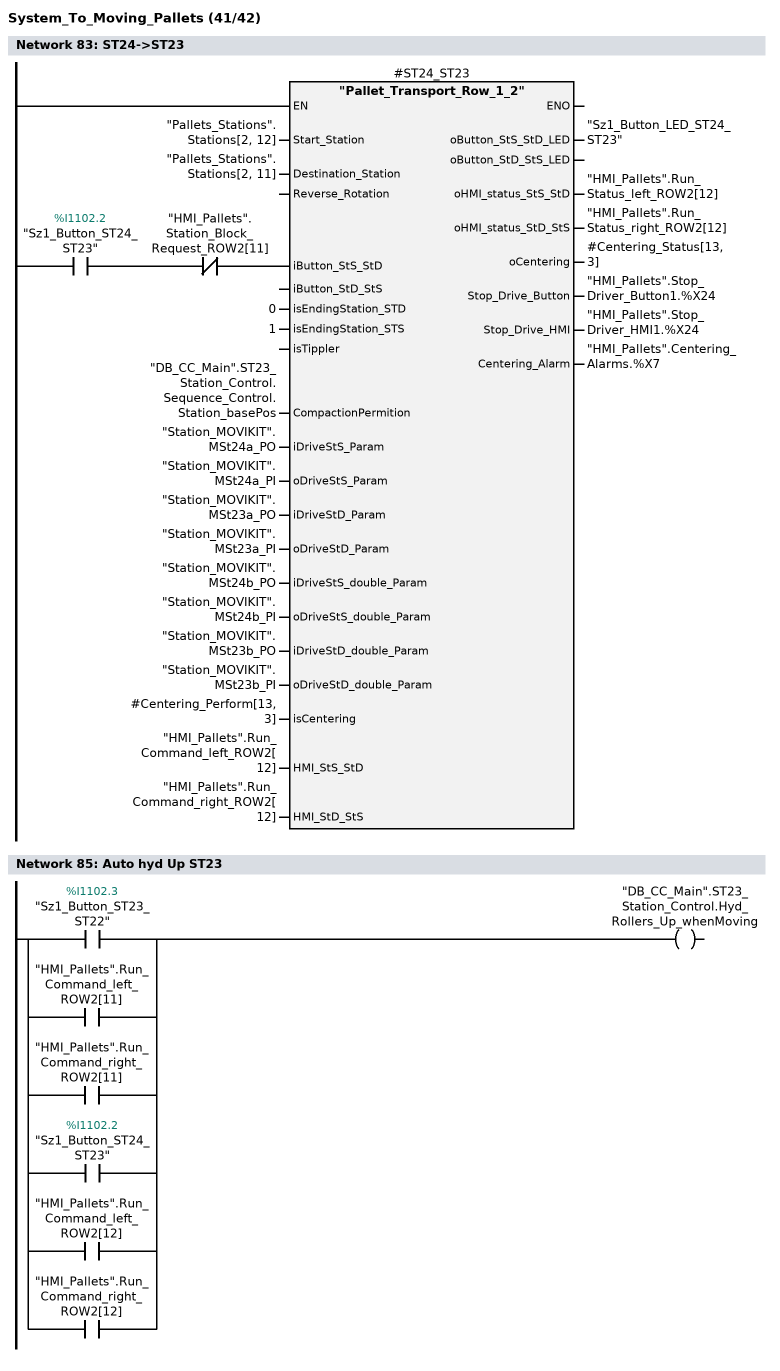
   RUNG wire#powerrail
      #ST24_ST23(iButton_StS_StD := wire#w1, Start_Station := "Pallets_Stations".Stations[2, 12], Destination_Station := "Pallets_Stations".Stations[2, 11], Reverse_Rotation :=, iButton_StD_StS :=, isEndingStation_STD := 0, isEndingStation_STS := 1, isTippler :=, CompactionPermition := "DB_CC_Main".ST23_Station_Control.Sequence_Control.Station_basePos, iDriveStS_Param := "Station_MOVIKIT".MSt24a_PO, oDriveStS_Param := "Station_MOVIKIT".MSt24a_PI, iDriveStD_Param := "Station_MOVIKIT".MSt23a_PO, oDriveStD_Param := "Station_MOVIKIT".MSt23a_PI, iDriveStS_double_Param := "Station_MOVIKIT".MSt24b_PO, oDriveStS_double_Param := "Station_MOVIKIT".MSt24b_PI, iDriveStD_double_Param := "Station_MOVIKIT".MSt23b_PO, oDriveStD_double_Param := "Station_MOVIKIT".MSt23b_PI, isCentering := #Centering_Perform[13, 3], HMI_StS_StD := "HMI_Pallets".Run_Command_left_ROW2[12], HMI_StD_StS := "HMI_Pallets".Run_Command_right_ROW2[12], oButton_StS_StD_LED => "Sz1_Button_LED_ST24_ST23", oButton_StD_StS_LED =>, oHMI_status_StS_StD => "HMI_Pallets".Run_Status_left_ROW2[12], oHMI_status_StD_StS => "HMI_Pallets".Run_Status_right_ROW2[12], oCentering => #Centering_Status[13, 3], Stop_Drive_Button => "HMI_Pallets".Stop_Driver_Button1.%X24, Stop_Drive_HMI => "HMI_Pallets".Stop_Driver_HMI1.%X24, Centering_Alarm => "HMI_Pallets".Centering_Alarms.%X7)
   END_RUNG
   RUNG wire#powerrail
      Contact( "Sz1_Button_ST24_ST23" )
      I_Contact( "HMI_Pallets".Station_Block_Request_ROW2[11] )
   END_RUNG wire#w1
   // the same network as SCL:
   #ST24_ST23(Start_Station := "Pallets_Stations".Stations[2, 12],   // "Pallet_Transport_Row_1_2"
              Destination_Station := "Pallets_Stations".Stations[2, 11],
              iButton_StS_StD := "Sz1_Button_ST24_ST23" AND NOT "HMI_Pallets".Station_Block_Request_ROW2[11],
              isEndingStation_STD := 0,
              isEndingStation_STS := 1,
              CompactionPermition := "DB_CC_Main".ST23_Station_Control.Sequence_Control.Station_basePos,
              iDriveStS_Param := "Station_MOVIKIT".MSt24a_PO,
              oDriveStS_Param := "Station_MOVIKIT".MSt24a_PI,
              iDriveStD_Param := "Station_MOVIKIT".MSt23a_PO,
              oDriveStD_Param := "Station_MOVIKIT".MSt23a_PI,
              iDriveStS_double_Param := "Station_MOVIKIT".MSt24b_PO,
              oDriveStS_double_Param := "Station_MOVIKIT".MSt24b_PI,
              iDriveStD_double_Param := "Station_MOVIKIT".MSt23b_PO,
              oDriveStD_double_Param := "Station_MOVIKIT".MSt23b_PI,
              isCentering := #Centering_Perform[13, 3],
              HMI_StS_StD := "HMI_Pallets".Run_Command_left_ROW2[12],
              HMI_StD_StS := "HMI_Pallets".Run_Command_right_ROW2[12],
              oButton_StS_StD_LED => "Sz1_Button_LED_ST24_ST23",
              oHMI_status_StS_StD => "HMI_Pallets".Run_Status_left_ROW2[12],
              oHMI_status_StD_StS => "HMI_Pallets".Run_Status_right_ROW2[12],
              oCentering => #Centering_Status[13, 3],
              Stop_Drive_Button => "HMI_Pallets".Stop_Driver_Button1.%X24,
              Stop_Drive_HMI => "HMI_Pallets".Stop_Driver_HMI1.%X24,
              Centering_Alarm => "HMI_Pallets".Centering_Alarms.%X7);
END_REGION

REGION Network 84 (SCL): Reset centering status of Tippler
   IF ("Station_MOVIKIT".MSt1_PO.x_Bit_1_Enable_Application_Stop OR "Station_MOVIKIT".MSt1a_PO.x_Bit_1_Enable_Application_Stop) AND #oCeterTippler THEN
       #Reset_Centering_Tippler := 1;
   ELSE
       #Reset_Centering_Tippler := 0;
   END_IF;
END_REGION

REGION Network 85: Auto hyd Up ST23
   RUNG wire#powerrail
      Contact( "Sz1_Button_ST23_ST22" )
      wire#w1
      Coil( "DB_CC_Main".ST23_Station_Control.Hyd_Rollers_Up_whenMoving )
   END_RUNG
   RUNG wire#powerrail
      Contact( "HMI_Pallets".Run_Command_left_ROW2[11] )
   END_RUNG wire#w1
   RUNG wire#powerrail
      Contact( "HMI_Pallets".Run_Command_right_ROW2[11] )
   END_RUNG wire#w1
   RUNG wire#powerrail
      Contact( "Sz1_Button_ST24_ST23" )
   END_RUNG wire#w1
   RUNG wire#powerrail
      Contact( "HMI_Pallets".Run_Command_left_ROW2[12] )
   END_RUNG wire#w1
   RUNG wire#powerrail
      Contact( "HMI_Pallets".Run_Command_right_ROW2[12] )
   END_RUNG wire#w1
   // the same network as SCL:
   "DB_CC_Main".ST23_Station_Control.Hyd_Rollers_Up_whenMoving := "Sz1_Button_ST23_ST22" OR "HMI_Pallets".Run_Command_left_ROW2[11] OR "HMI_Pallets".Run_Command_right_ROW2[11] OR "Sz1_Button_ST24_ST23" OR "HMI_Pallets".Run_Command_left_ROW2[12] OR "HMI_Pallets".Run_Command_right_ROW2[12];
END_REGION

REGION Network 86: Auto hyd Up ST24
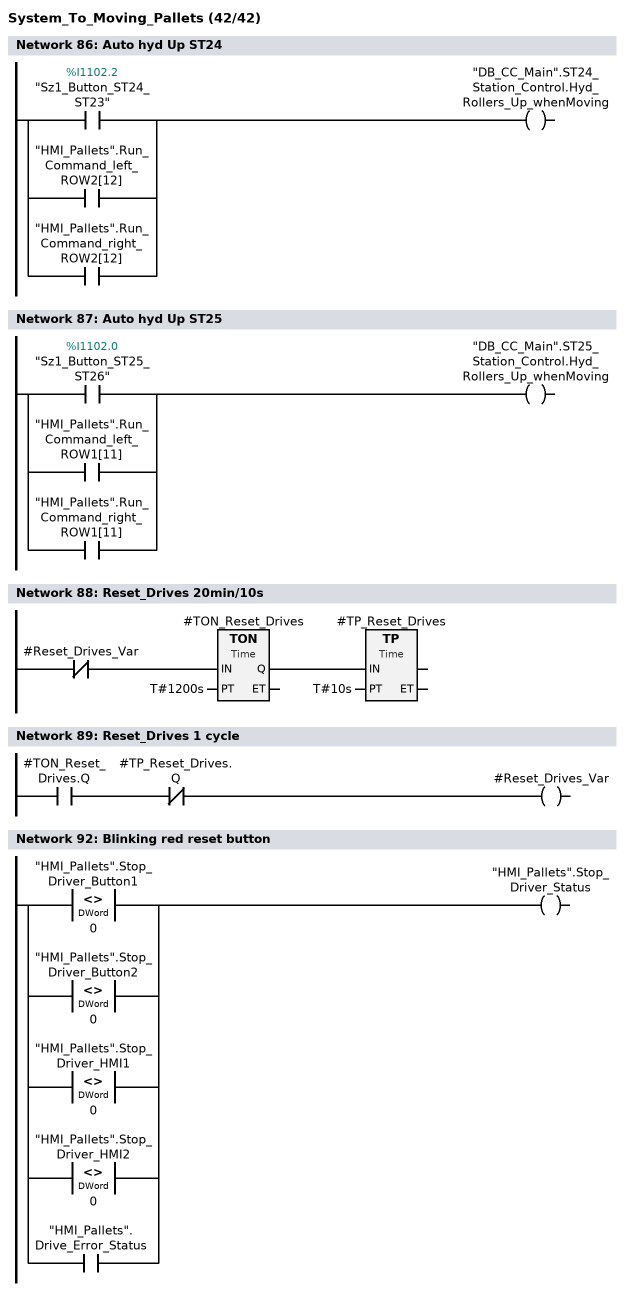
   RUNG wire#powerrail
      Contact( "Sz1_Button_ST24_ST23" )
      wire#w1
      Coil( "DB_CC_Main".ST24_Station_Control.Hyd_Rollers_Up_whenMoving )
   END_RUNG
   RUNG wire#powerrail
      Contact( "HMI_Pallets".Run_Command_left_ROW2[12] )
   END_RUNG wire#w1
   RUNG wire#powerrail
      Contact( "HMI_Pallets".Run_Command_right_ROW2[12] )
   END_RUNG wire#w1
   // the same network as SCL:
   "DB_CC_Main".ST24_Station_Control.Hyd_Rollers_Up_whenMoving := "Sz1_Button_ST24_ST23" OR "HMI_Pallets".Run_Command_left_ROW2[12] OR "HMI_Pallets".Run_Command_right_ROW2[12];
END_REGION

REGION Network 87: Auto hyd Up ST25
   RUNG wire#powerrail
      Contact( "Sz1_Button_ST25_ST26" )
      wire#w1
      Coil( "DB_CC_Main".ST25_Station_Control.Hyd_Rollers_Up_whenMoving )
   END_RUNG
   RUNG wire#powerrail
      Contact( "HMI_Pallets".Run_Command_left_ROW1[11] )
   END_RUNG wire#w1
   RUNG wire#powerrail
      Contact( "HMI_Pallets".Run_Command_right_ROW1[11] )
   END_RUNG wire#w1
   // the same network as SCL:
   "DB_CC_Main".ST25_Station_Control.Hyd_Rollers_Up_whenMoving := "Sz1_Button_ST25_ST26" OR "HMI_Pallets".Run_Command_left_ROW1[11] OR "HMI_Pallets".Run_Command_right_ROW1[11];
END_REGION

REGION Network 88: Reset_Drives 20min/10s
   RUNG wire#powerrail
      I_Contact( #Reset_Drives_Var )
      { S7_Templates := "time_type := Time" } #TON_Reset_Drives.TON(pt := T#1200s, et =>)
      { S7_Templates := "time_type := Time" } #TP_Reset_Drives.TP(pt := T#10s, et =>)
   END_RUNG
   // the same network as SCL:
   #TON_Reset_Drives(IN := NOT #Reset_Drives_Var, PT := T#1200s);   // TON
   #TP_Reset_Drives(IN := #TON_Reset_Drives.Q, PT := T#10s);   // TP
END_REGION

REGION Network 89: Reset_Drives 1 cycle
   RUNG wire#powerrail
      Contact( #TON_Reset_Drives.Q )
      I_Contact( #TP_Reset_Drives.Q )
      Coil( #Reset_Drives_Var )
   END_RUNG
   // the same network as SCL:
   #Reset_Drives_Var := #TON_Reset_Drives.Q AND NOT #TP_Reset_Drives.Q;
END_REGION

REGION Network 90 (SCL): Select Pallet
   FOR #i := 1 TO 24 DO
       IF #i = "HMI_Pallets".Number_Of_Pallet THEN
           "Pallets_Stations".Pallets[#i].IsSelected := 1;
       ELSE
           "Pallets_Stations".Pallets[#i].IsSelected := 0;
       END_IF;
   END_FOR;
END_REGION

REGION Network 91 (SCL): Cyclic reset drive command
   IF #Reset_Drives_Var OR "HMI_Test_DB".HMI_Connection_Alarm THEN

       FOR #i := 1 TO 12 DO
           "HMI_Pallets".Run_Command_left_ROW1[#i] := FALSE;
           "HMI_Pallets".Run_Command_left_ROW2[#i] := FALSE;
           "HMI_Pallets".Run_Command_left_ROW4[#i] := FALSE;
           "HMI_Pallets".Run_Command_right_ROW1[#i] := FALSE;
           "HMI_Pallets".Run_Command_right_ROW2[#i] := FALSE;
           "HMI_Pallets".Run_Command_right_ROW4[#i] := FALSE;
       END_FOR;
   END_IF;
END_REGION

REGION Network 92: Blinking red reset button
   RUNG wire#powerrail
      { S7_Templates := "SrcType := DWord" } NE_Contact(in1 := "HMI_Pallets".Stop_Driver_Button1, in2 := 0)
      wire#w1
      Coil( "HMI_Pallets".Stop_Driver_Status )
   END_RUNG
   RUNG wire#powerrail
      { S7_Templates := "SrcType := DWord" } NE_Contact(in1 := "HMI_Pallets".Stop_Driver_Button2, in2 := 0)
   END_RUNG wire#w1
   RUNG wire#powerrail
      { S7_Templates := "SrcType := DWord" } NE_Contact(in1 := "HMI_Pallets".Stop_Driver_HMI1, in2 := 0)
   END_RUNG wire#w1
   RUNG wire#powerrail
      { S7_Templates := "SrcType := DWord" } NE_Contact(in1 := "HMI_Pallets".Stop_Driver_HMI2, in2 := 0)
   END_RUNG wire#w1
   RUNG wire#powerrail
      Contact( "HMI_Pallets".Drive_Error_Status )
   END_RUNG wire#w1
   // the same network as SCL:
   "HMI_Pallets".Stop_Driver_Status := ("HMI_Pallets".Stop_Driver_Button1 <> 0) OR ("HMI_Pallets".Stop_Driver_Button2 <> 0) OR ("HMI_Pallets".Stop_Driver_HMI1 <> 0) OR ("HMI_Pallets".Stop_Driver_HMI2 <> 0) OR "HMI_Pallets".Drive_Error_Status;
END_REGION

REGION Network 93 (SCL): W1-W2-W4 Command Run: TImeout/Multichoice RESET
   REGION W1 Reset
       // Timer ON when Command_Run_W1 = 1
       #tComm_W1(IN := "HMI_Pallets".Command_Run_W1,
                 PT := T#2m);

       // Reset after 2m
       IF #tComm_W1.Q THEN
           "HMI_Pallets".Command_Run_W1 := FALSE;
       END_IF;

   END_REGION

   REGION W2 Reset
       // Timer ON when Command_Run_W2 = 1
       #tComm_W2(IN := "HMI_Pallets".Command_Run_W2,
                 PT := T#2m);

       // Reset after 2m
       IF #tComm_W2.Q THEN
           "HMI_Pallets".Command_Run_W2 := FALSE;
       END_IF;

   END_REGION


   REGION W4 Reset
       // Timer ON when Command_Run_W4 = 1
       #tComm_W4(IN := "HMI_Pallets".Command_Run_W4,
                 PT := T#2m);

       // Reset after 2m
       IF #tComm_W4.Q THEN
           "HMI_Pallets".Command_Run_W4 := FALSE;
       END_IF;

   END_REGION

   //TO DO change W1 & W2 to W1_2 
   IF (
       ("HMI_Pallets".Command_Run_W1 AND "HMI_Pallets".Command_Run_W2) OR
       ("HMI_Pallets".Command_Run_W1 AND "HMI_Pallets".Command_Run_W4) OR
       ("HMI_Pallets".Command_Run_W2 AND "HMI_Pallets".Command_Run_W4)
       ) THEN

       "HMI_Pallets".Command_Run_W1 := FALSE;
       "HMI_Pallets".Command_Run_W2 := FALSE;
       "HMI_Pallets".Command_Run_W4 := FALSE;

   END_IF;
END_REGION

REGION Network 94 (SCL): Station Block Request: Global Button RESET / Block Active CHECK
   // REGION BLOCK_RESET - Reset Block Request
   // REGION ANY_STATION_BLOCK_ACTIVE - Check if any Block is Active (HMI Color Purposes)
   REGION BLOCK_RESET

       IF "HMI_Pallets".Reset_Station_Block_Request THEN

           FOR #Reset_Stations_Index := 1 TO 12 DO
               "HMI_Pallets".Station_Block_Request_ROW1[#Reset_Stations_Index] := FALSE;
               "HMI_Pallets".Station_Block_Request_ROW2[#Reset_Stations_Index] := FALSE;
               "HMI_Pallets".Station_Block_Request_ROW4[#Reset_Stations_Index] := FALSE;
           END_FOR;

           "HMI_Pallets".Reset_Station_Block_Request := FALSE;

       END_IF;

   END_REGION


   REGION ANY_STATION_BLOCK_ACTIVE
       "HMI_Pallets".Any_Station_Block_ACTIVE := FALSE;

       FOR #Block_Check_Index := 1 TO 12 DO

              "HMI_Pallets".Any_Station_Block_ACTIVE :="HMI_Pallets".Any_Station_Block_ACTIVE

               OR "HMI_Pallets".Station_Block_Request_ROW1[#Block_Check_Index]
               OR "HMI_Pallets".Station_Block_Request_ROW2[#Block_Check_Index]
               OR "HMI_Pallets".Station_Block_Request_ROW4[#Block_Check_Index];

       END_FOR;

   END_REGION
END_REGION

REGION Network 95: #################################################################
END_REGION
END_FUNCTION_BLOCK

FUNCTION "Initialisations" : Void
{ S7_Optimized_Access := 'TRUE' }
VERSION : 0.1
   VAR_TEMP 
      i : Int;
      j : Int;
   END_VAR


BEGIN
	REGION Stations_Sensors
	    
	    // row 1
	    
	    "Pallets_Stations".Stations[1, 1].SensorA := "Sz5_ST35_SenA";
	    "Pallets_Stations".Stations[1, 1].SensorB := "Sz5_ST35_SenB";
	    "Pallets_Stations".Stations[1, 1].SensorC := "Sz5_ST35_SenC";
	    "Pallets_Stations".Stations[1, 1].SensorD := "Sz5_ST35_SenD";
	    
	    "Pallets_Stations".Stations[1, 2].SensorA := "Sz5_ST34_SenA";
	    "Pallets_Stations".Stations[1, 2].SensorB := "Sz5_ST34_SenB";
	    "Pallets_Stations".Stations[1, 2].SensorC := "Sz5_ST34_SenC";
	    "Pallets_Stations".Stations[1, 2].SensorD := "Sz5_ST34_SenD";
	    
	    "Pallets_Stations".Stations[1, 3].SensorA := "Sz4_ST33_SenA";
	    "Pallets_Stations".Stations[1, 3].SensorB := "Sz4_ST33_SenB";
	    "Pallets_Stations".Stations[1, 3].SensorC := "Sz4_ST33_SenC";
	    "Pallets_Stations".Stations[1, 3].SensorD := "Sz4_ST33_SenD";
	    
	    "Pallets_Stations".Stations[1, 4].SensorA := "Sz4_ST32_SenA";
	    "Pallets_Stations".Stations[1, 4].SensorB := "Sz4_ST32_SenB";
	    "Pallets_Stations".Stations[1, 4].SensorC := "Sz4_ST32_SenC";
	    "Pallets_Stations".Stations[1, 4].SensorD := "Sz4_ST32_SenD";
	    
	    "Pallets_Stations".Stations[1, 5].SensorA := "Sz3_ST31_SenA";
	    "Pallets_Stations".Stations[1, 5].SensorB := "Sz3_ST31_SenB";
	    "Pallets_Stations".Stations[1, 5].SensorC := "Sz3_ST31_SenC";
	    "Pallets_Stations".Stations[1, 5].SensorD := "Sz3_ST31_SenD";
	    
	    "Pallets_Stations".Stations[1, 6].SensorA := "Sz3_ST30_SenA";
	    "Pallets_Stations".Stations[1, 6].SensorB := "Sz3_ST30_SenB";
	    "Pallets_Stations".Stations[1, 6].SensorC := "Sz3_ST30_SenC";
	    "Pallets_Stations".Stations[1, 6].SensorD := "Sz3_ST30_SenD";
	    
	    "Pallets_Stations".Stations[1, 7].SensorA := "Sz3_ST29_SenA";
	    "Pallets_Stations".Stations[1, 7].SensorB := "Sz3_ST29_SenB";
	    "Pallets_Stations".Stations[1, 7].SensorC := "Sz3_ST29_SenC";
	    "Pallets_Stations".Stations[1, 7].SensorD := "Sz3_ST29_SenD";
	    
	    "Pallets_Stations".Stations[1, 8].SensorA := "Sz2_ST28_SenA";
	    "Pallets_Stations".Stations[1, 8].SensorB := "Sz2_ST28_SenB";
	    "Pallets_Stations".Stations[1, 8].SensorC := "Sz2_ST28_SenC";
	    "Pallets_Stations".Stations[1, 8].SensorD := "Sz2_ST28_SenD";
	    
	    "Pallets_Stations".Stations[1, 9].SensorA := "Sz2_ST27_SenA";
	    "Pallets_Stations".Stations[1, 9].SensorB := "Sz2_ST27_SenB";
	    "Pallets_Stations".Stations[1, 9].SensorC := "Sz2_ST27_SenC";
	    "Pallets_Stations".Stations[1, 9].SensorD := "Sz2_ST27_SenD";
	    
	    "Pallets_Stations".Stations[1, 10].SensorA := "Sz1_St26_SenA";
	    "Pallets_Stations".Stations[1, 10].SensorB := "Sz1_St26_SenB";
	    "Pallets_Stations".Stations[1, 10].SensorC := "Sz1_St26_SenC";
	    "Pallets_Stations".Stations[1, 10].SensorD := "Sz1_St26_SenD";
	    
	    "Pallets_Stations".Stations[1, 11].SensorA := "Sz1_St25_SenA";
	    "Pallets_Stations".Stations[1, 11].SensorB := "Sz1_St25_SenB";
	    "Pallets_Stations".Stations[1, 11].SensorC := "Sz1_St25_SenC";
	    "Pallets_Stations".Stations[1, 11].SensorD := "Sz1_St25_SenD";
	    
	    //row 2
	    
	    "Pallets_Stations".Stations[2, 2].SensorA := "Sz5_ST01_SenA";
	    "Pallets_Stations".Stations[2, 2].SensorB := "Sz5_ST01_SenB";
	    "Pallets_Stations".Stations[2, 2].SensorC := "Sz5_ST01_SenC";
	    "Pallets_Stations".Stations[2, 2].SensorD := "Sz5_ST01_SenD";
	    
	    "Pallets_Stations".Stations[2, 1].SensorA := "Sz5_ST02_SenA";
	    "Pallets_Stations".Stations[2, 1].SensorB := "Sz5_ST02_SenB";
	    "Pallets_Stations".Stations[2, 1].SensorC := "Sz5_ST02_SenC";
	    "Pallets_Stations".Stations[2, 1].SensorD := "Sz5_ST02_SenD";
	    
	    "Pallets_Stations".Stations[2, 3].SensorA := "Sz5_ST38_SenA";
	    "Pallets_Stations".Stations[2, 3].SensorB := "Sz5_ST38_SenB";
	    "Pallets_Stations".Stations[2, 3].SensorC := "Sz5_ST38_SenC";
	    "Pallets_Stations".Stations[2, 3].SensorD := "Sz5_ST38_SenD";
	    
	    "Pallets_Stations".Stations[2, 4].SensorA := "Sz4_ST36_SenA";
	    "Pallets_Stations".Stations[2, 4].SensorB := "Sz4_ST36_SenB";
	    "Pallets_Stations".Stations[2, 4].SensorC := "Sz4_ST36_SenC";
	    "Pallets_Stations".Stations[2, 4].SensorD := "Sz4_ST36_SenD";
	    
	    "Pallets_Stations".Stations[2, 5].SensorA := "Sz4_ST37_SenA";
	    "Pallets_Stations".Stations[2, 5].SensorB := "Sz4_ST37_SenB";
	    "Pallets_Stations".Stations[2, 5].SensorC := "Sz4_ST37_SenC";
	    "Pallets_Stations".Stations[2, 5].SensorD := "Sz4_ST37_SenD";
	    
	    "Pallets_Stations".Stations[2, 6].SensorA := "Sz3_ST18_SenA";
	    "Pallets_Stations".Stations[2, 6].SensorB := "Sz3_ST18_SenB";
	    "Pallets_Stations".Stations[2, 6].SensorC := "Sz3_ST18_SenC";
	    "Pallets_Stations".Stations[2, 6].SensorD := "Sz3_ST18_SenD";
	    
	    "Pallets_Stations".Stations[2, 7].SensorA := "Sz3_ST19_SenA";
	    "Pallets_Stations".Stations[2, 7].SensorB := "Sz3_ST19_SenB";
	    "Pallets_Stations".Stations[2, 7].SensorC := "Sz3_ST19_SenC";
	    "Pallets_Stations".Stations[2, 7].SensorD := "Sz3_ST19_SenD";
	    
	    "Pallets_Stations".Stations[2, 8].SensorA := "Sz3_ST20_SenA";
	    "Pallets_Stations".Stations[2, 8].SensorB := "Sz3_ST20_SenB";
	    "Pallets_Stations".Stations[2, 8].SensorC := "Sz3_ST20_SenC";
	    "Pallets_Stations".Stations[2, 8].SensorD := "Sz3_ST20_SenD";
	    
	    "Pallets_Stations".Stations[2, 9].SensorA := "Sz2_ST21_SenA";
	    "Pallets_Stations".Stations[2, 9].SensorB := "Sz2_ST21_SenB";
	    "Pallets_Stations".Stations[2, 9].SensorC := "Sz2_ST21_SenC";
	    "Pallets_Stations".Stations[2, 9].SensorD := "Sz2_ST21_SenD";
	    
	    "Pallets_Stations".Stations[2, 10].SensorA := "Sz2_ST22_SenA";
	    "Pallets_Stations".Stations[2, 10].SensorB := "Sz2_ST22_SenB";
	    "Pallets_Stations".Stations[2, 10].SensorC := "Sz2_ST22_SenC";
	    "Pallets_Stations".Stations[2, 10].SensorD := "Sz2_ST22_SenD";
	    
	    "Pallets_Stations".Stations[2, 11].SensorA := "Sz1_St23_SenA";
	    "Pallets_Stations".Stations[2, 11].SensorB := "Sz1_St23_SenB";
	    "Pallets_Stations".Stations[2, 11].SensorC := "Sz1_St23_SenC";
	    "Pallets_Stations".Stations[2, 11].SensorD := "Sz1_St23_SenD";
	    
	    "Pallets_Stations".Stations[2, 12].SensorA := "Sz1_St24_SenA";
	    "Pallets_Stations".Stations[2, 12].SensorB := "Sz1_St24_SenB";
	    "Pallets_Stations".Stations[2, 12].SensorC := "Sz1_St24_SenC";
	    "Pallets_Stations".Stations[2, 12].SensorD := "Sz1_St24_SenD";
	    
	    // row 3
	    
	    "Pallets_Stations".Stations[3, 1].SensorA := "Sz7_ST03_SenA";
	    "Pallets_Stations".Stations[3, 1].SensorB := "Sz7_ST03_SenB";
	    "Pallets_Stations".Stations[3, 1].SensorC := "Sz7_ST03_SenC";
	    "Pallets_Stations".Stations[3, 1].SensorD := "Sz7_ST03_SenD";
	    
	    "Pallets_Stations".Stations[3, 11].SensorA := "Sz11_ST17_SenA";
	    "Pallets_Stations".Stations[3, 11].SensorB := "Sz11_ST17_SenB";
	    "Pallets_Stations".Stations[3, 11].SensorC := "Sz11_ST17_SenC";
	    "Pallets_Stations".Stations[3, 11].SensorD := "Sz11_ST17_SenD";
	    
	    // row 4
	    
	    "Pallets_Stations".Stations[4, 1].SensorA := "Sz7_ST04_SenA";
	    "Pallets_Stations".Stations[4, 1].SensorB := "Sz7_ST04_SenB";
	    "Pallets_Stations".Stations[4, 1].SensorC := "Sz7_ST04_SenC";
	    "Pallets_Stations".Stations[4, 1].SensorD := "Sz7_ST04_SenD";
	    
	    "Pallets_Stations".Stations[4, 2].SensorA := "Sz7_ST05_SenA";
	    "Pallets_Stations".Stations[4, 2].SensorB := "Sz7_ST05_SenB";
	    "Pallets_Stations".Stations[4, 2].SensorC := "Sz7_ST05_SenC";
	    "Pallets_Stations".Stations[4, 2].SensorD := "Sz7_ST05_SenD";
	    
	    "Pallets_Stations".Stations[4, 3].SensorA := "Sz8_ST06_SenA";
	    "Pallets_Stations".Stations[4, 3].SensorB := "Sz8_ST06_SenB";
	    "Pallets_Stations".Stations[4, 3].SensorC := "Sz8_ST06_SenC";
	    "Pallets_Stations".Stations[4, 3].SensorD := "Sz8_ST06_SenD";
	    
	    "Pallets_Stations".Stations[4, 4].SensorA := "Sz8_ST07_SenA";
	    "Pallets_Stations".Stations[4, 4].SensorB := "Sz8_ST07_SenB";
	    "Pallets_Stations".Stations[4, 4].SensorC := "Sz8_ST07_SenC";
	    "Pallets_Stations".Stations[4, 4].SensorD := "Sz8_ST07_SenD";
	    
	    "Pallets_Stations".Stations[4, 5].SensorA := "Sz8_ST08_SenA";
	    "Pallets_Stations".Stations[4, 5].SensorB := "Sz8_ST08_SenB";
	    "Pallets_Stations".Stations[4, 5].SensorC := "Sz8_ST08_SenC";
	    "Pallets_Stations".Stations[4, 5].SensorD := "Sz8_ST08_SenD";
	    
	    "Pallets_Stations".Stations[4, 6].SensorA := "Sz9_ST09_SenA";
	    "Pallets_Stations".Stations[4, 6].SensorB := "Sz9_ST09_SenB";
	    "Pallets_Stations".Stations[4, 6].SensorC := "Sz9_ST09_SenC";
	    "Pallets_Stations".Stations[4, 6].SensorD := "Sz9_ST09_SenD";
	    
	    "Pallets_Stations".Stations[4, 7].SensorA := "Sz9_ST10_SenA";
	    "Pallets_Stations".Stations[4, 7].SensorB := "Sz9_ST10_SenB";
	    "Pallets_Stations".Stations[4, 7].SensorC := "Sz9_ST10_SenC";
	    "Pallets_Stations".Stations[4, 7].SensorD := "Sz9_ST10_SenD";
	    
	    "Pallets_Stations".Stations[4, 8].SensorA := "Sz10_ST11_SenA";
	    "Pallets_Stations".Stations[4, 8].SensorB := "Sz10_ST11_SenB";
	    "Pallets_Stations".Stations[4, 8].SensorC := "Sz10_ST11_SenC";
	    "Pallets_Stations".Stations[4, 8].SensorD := "Sz10_ST11_SenD";
	    
	    "Pallets_Stations".Stations[4, 9].SensorA := "Sz10_ST12_SenA";
	    "Pallets_Stations".Stations[4, 9].SensorB := "Sz10_ST12_SenB";
	    "Pallets_Stations".Stations[4, 9].SensorC := "Sz10_ST12_SenC";
	    "Pallets_Stations".Stations[4, 9].SensorD := "Sz10_ST12_SenD";
	    
	    "Pallets_Stations".Stations[4, 10].SensorA := "Sz11_ST13_SenA";
	    "Pallets_Stations".Stations[4, 10].SensorB := "Sz11_ST13_SenB";
	    "Pallets_Stations".Stations[4, 10].SensorC := "Sz11_ST13_SenC";
	    "Pallets_Stations".Stations[4, 10].SensorD := "Sz11_ST13_SenD";
	    
	    "Pallets_Stations".Stations[4, 11].SensorA := "Sz11_ST14_SenA";
	    "Pallets_Stations".Stations[4, 11].SensorB := "Sz11_ST14_SenB";
	    "Pallets_Stations".Stations[4, 11].SensorC := "Sz11_ST14_SenC";
	    "Pallets_Stations".Stations[4, 11].SensorD := "Sz11_ST14_SenD";
	    
	END_REGION
	
	REGION Station_Status
	    
	    FOR #i := 1 TO 4 DO
	        FOR #j := 1 TO 12 DO
	            // CentralShifter
	            IF (#i = 3 AND (#j >= 2 AND #j <= 10)) OR
	                ((#i = 1 OR #i = 3 OR #i = 4) AND #j = 12) THEN // Last column
	                "Pallets_Stations".Stations[#i, #j].IsOccupied := TRUE;
	                "Pallets_Stations".Stations[#i, #j].IsEmpty := FALSE;
	                // All sensors are True
	            ELSIF "Pallets_Stations".Stations[#i, #j].SensorA AND
	                "Pallets_Stations".Stations[#i, #j].SensorB AND
	                "Pallets_Stations".Stations[#i, #j].SensorC AND
	                "Pallets_Stations".Stations[#i, #j].SensorD THEN
	                "Pallets_Stations".Stations[#i, #j].IsOccupied := TRUE;
	                "Pallets_Stations".Stations[#i, #j].IsEmpty := FALSE;
	                // All sensors are False
	            ELSIF NOT "Pallets_Stations".Stations[#i, #j].SensorA AND
	                NOT "Pallets_Stations".Stations[#i, #j].SensorB AND
	                NOT "Pallets_Stations".Stations[#i, #j].SensorC AND
	                NOT "Pallets_Stations".Stations[#i, #j].SensorD THEN
	                "Pallets_Stations".Stations[#i, #j].IsEmpty := TRUE;
	                "Pallets_Stations".Stations[#i, #j].IsOccupied := FALSE;
	            ELSE
	                // Unknown state
	                "Pallets_Stations".Stations[#i, #j].IsEmpty := FALSE;
	                "Pallets_Stations".Stations[#i, #j].IsOccupied := FALSE;
	            END_IF;
	            
	            CASE #i OF
	                1:
	                    "CopyStationBase"(InStation := "Pallets_Stations".Stations[#i, #j],
	                                      OutStation => "Pallets_Stations".Stations_ROW1[#j]);
	                2:
	                    "CopyStationBase"(InStation := "Pallets_Stations".Stations[#i, #j],
	                                      OutStation => "Pallets_Stations".Stations_ROW2[#j]);
	                3:
	                    "CopyStationBase"(InStation := "Pallets_Stations".Stations[#i, #j],
	                                      OutStation => "Pallets_Stations".Stations_ROW3[#j]);
	                4:
	                    "CopyStationBase"(InStation := "Pallets_Stations".Stations[#i, #j],
	                                      OutStation => "Pallets_Stations".Stations_ROW4[#j]);
	            END_CASE;
	        END_FOR;
	    END_FOR;
	    
	END_REGION
END_FUNCTION

FUNCTION "CopyStationBase" : Void
{ S7_Optimized_Access := 'TRUE' }
VERSION : 0.1
   VAR_INPUT 
      InStation : "Station";
   END_VAR

   VAR_OUTPUT 
      OutStation : "StationLight";
   END_VAR


BEGIN
	#OutStation.SensorA := #InStation.SensorA;
	#OutStation.SensorB := #InStation.SensorB;
	#OutStation.SensorC := #InStation.SensorC;
	#OutStation.SensorD := #InStation.SensorD;
	#OutStation.IsEmpty := #InStation.IsEmpty;
	#OutStation.IsOccupied := #InStation.IsOccupied;
	
END_FUNCTION

FUNCTION "Drivers_To_Move_Pallet" : Void   // FC5, LAD
{ S7_Optimized_Access := 'TRUE' }
// stored: SetENOAutomatically false
   VAR_INPUT
      HW_Driver : HW_IO;
      Reset : Bool;
   END_VAR
   VAR_IN_OUT
      iDrive_Param : "SEW_MOVIKIT_VelocityDrive_SETPOINTS_V2.1";
      oDrive_Param : "SEW_MOVIKIT_VelocityDrive_STATUS_V2.1";
   END_VAR
   VAR_TEMP
      Communication_OK : Bool;
   END_VAR
BEGIN

REGION Network 1
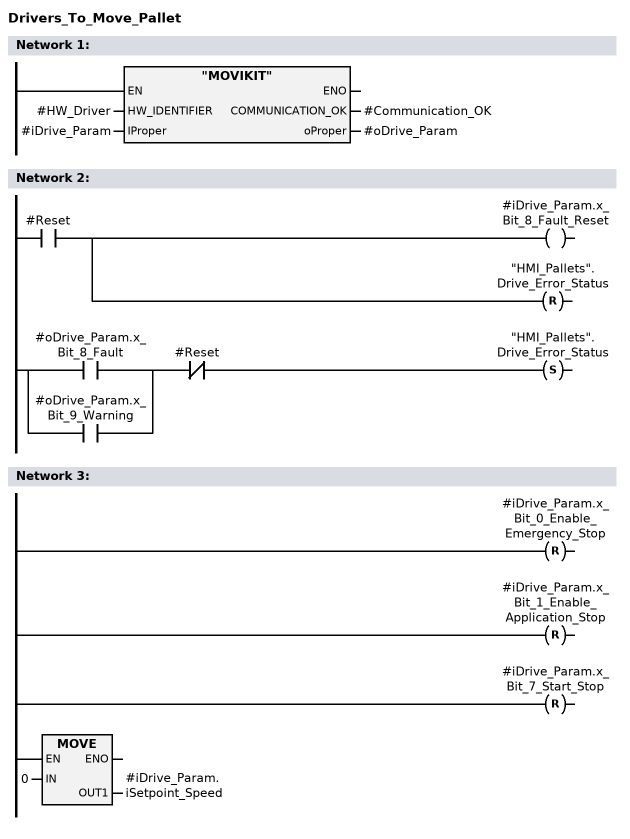
   RUNG wire#powerrail
      "MOVIKIT"(HW_IDENTIFIER := #HW_Driver, IProper := #iDrive_Param, COMMUNICATION_OK => #Communication_OK, oProper => #oDrive_Param)
   END_RUNG
   // the same network as SCL:
   "MOVIKIT"(HW_IDENTIFIER := #HW_Driver,
             IProper := #iDrive_Param,
             COMMUNICATION_OK => #Communication_OK,
             oProper => #oDrive_Param);
END_REGION

REGION Network 2
   RUNG wire#powerrail
      Contact( #Reset )
      wire#w1
      Coil( #iDrive_Param.x_Bit_8_Fault_Reset )
   END_RUNG
   RUNG wire#w1
      R_Coil( "HMI_Pallets".Drive_Error_Status )
   END_RUNG
   RUNG wire#powerrail
      Contact( #oDrive_Param.x_Bit_8_Fault )
      wire#w2
      I_Contact( #Reset )
      S_Coil( "HMI_Pallets".Drive_Error_Status )
   END_RUNG
   RUNG wire#powerrail
      Contact( #oDrive_Param.x_Bit_9_Warning )
   END_RUNG wire#w2
   // the same network as SCL:
   #iDrive_Param.x_Bit_8_Fault_Reset := #Reset;
   IF #Reset THEN "HMI_Pallets".Drive_Error_Status := FALSE; END_IF;
   IF (#oDrive_Param.x_Bit_8_Fault OR #oDrive_Param.x_Bit_9_Warning) AND NOT #Reset THEN
       "HMI_Pallets".Drive_Error_Status := TRUE;
   END_IF;
END_REGION

REGION Network 3
   RUNG wire#powerrail
      R_Coil( #iDrive_Param.x_Bit_0_Enable_Emergency_Stop )
   END_RUNG
   RUNG wire#powerrail
      R_Coil( #iDrive_Param.x_Bit_1_Enable_Application_Stop )
   END_RUNG
   RUNG wire#powerrail
      R_Coil( #iDrive_Param.x_Bit_7_Start_Stop )
   END_RUNG
   RUNG wire#powerrail
      Move(in := 0, out1 => #iDrive_Param.iSetpoint_Speed)
   END_RUNG
   // the same network as SCL:
   #iDrive_Param.x_Bit_0_Enable_Emergency_Stop := FALSE;
   #iDrive_Param.x_Bit_1_Enable_Application_Stop := FALSE;
   #iDrive_Param.x_Bit_7_Start_Stop := FALSE;
   #iDrive_Param.iSetpoint_Speed := 0;
END_REGION
END_FUNCTION

FUNCTION "MOVIKIT" : Void
{ S7_Optimized_Access := 'FALSE' }
AUTHOR : SVSPASE
FAMILY : MOVIKIT
VERSION : 2.1
   VAR_INPUT 
      HW_IDENTIFIER : HW_IO;
      IProper : "SEW_MOVIKIT_VelocityDrive_SETPOINTS_V2.1";
   END_VAR

   VAR_OUTPUT 
      COMMUNICATION_OK : Bool;
      oProper : "SEW_MOVIKIT_VelocityDrive_STATUS_V2.1";
   END_VAR

   VAR_TEMP 
      PI : "SEW_MOVIKIT_VelocityDrive_STATUS_V2.1";
      PO : "SEW_MOVIKIT_VelocityDrive_SETPOINTS_V2.1";
      DPRD_RET_VAL : Int;
      DPWR_RET_VAL : Int;
   END_VAR


BEGIN
	(*This sample program only demonstrates the basic approach. We do not accept any legal or other liability for incorrect program functions and their consequences!
	
	The FC121 serves as a program module for controlling the MOVIKIT module "Velocity Drive+UDT" for the Generation C device series. With the help of the FC121,
	the converters can be controlled via PROFINET IO/PROFIBUS DP.
	
	Device & networks: To use this FC, a 5 PD slot must be configured.
	
	This FC uses the UDTs SEW_MOVIKIT_VelocityDrive_SETPOINTS_V2.1 and SEW_MOVIKIT_VelocityDrive_STATUS_V2.1. 
	Please make sure that these PLC data types are available in your TIA project.
	These UDTs can be copied from the original TIA sample project or from the MOVIKIT_Vel_&_Pos_UDTs_V2.x.al14 library.
	
	Attention Input "HW_Identifier":
	Assign the HW-Identifier of the 5 PD slot. S73xx/4xx:Change Data type from HW_IO to WORD;  Assign the peripheral address of the 5 PD slot
	*)
	
	//DPRD_DAT: Reading Consistent Data of a DP Standard Slave/PROFINET IO device
	#DPRD_RET_VAL := DPRD_DAT(LADDR := #HW_IDENTIFIER, RECORD => #PI);
	
	IF #DPRD_RET_VAL = 0 THEN //If no error occurs while the instruction is being executed...
	    #COMMUNICATION_OK := TRUE;
	    
	    //Mapping the signals of the Status word:
	    #oProper.x_Bit_0_Ready := #PI.x_Bit_0_Ready;
	    #oProper.x_Bit_1_STO_inactive := #PI.x_Bit_1_STO_inactive;
	    #oProper.x_Bit_2_Output_Stage_enabled := #PI.x_Bit_2_Output_Stage_enabled;
	    #oProper.x_Bit_3_Brake_released := #PI.x_Bit_3_Brake_released;
	    #oProper.x_Bit_4_Motor_turning :=#PI.x_Bit_4_Motor_turning;
	    #oProper.x_Bit_8_Fault := #PI.x_Bit_8_Fault;
	    #oProper.x_Bit_9_Warning := #PI.x_Bit_9_Warning;
	    #oProper.x_Bit_10_DriveTrain2_active := #PI.x_Bit_10_DriveTrain2_active;
	    #oProper.x_Bit_11_Setp_actual_speed_comp_signal_active := #PI.x_Bit_11_Setp_actual_speed_comp_signal_active;
	    #oProper.x_Bit_14_StandBy_Mode_active := #PI.x_Bit_14_StandBy_Mode_active;
	    #oProper.x_Bit_15_Heartbeat_OUT := #PI.x_Bit_15_Heartbeat_OUT;
	    
	    //Assign PI2..5
	    #oProper.iActual_Speed := #PI.iActual_Speed;
	    #oProper.wStatus_main_fault_sub_fault := #PI.wStatus_main_fault_sub_fault;
	    #oProper.bStatus_Fault := #oProper.wStatus_main_fault_sub_fault.%B1;
	    #oProper.bStatus_subFault := #oProper.wStatus_main_fault_sub_fault.%B0;
	    #oProper.iActual_Torque := #PI.iActual_Torque;
	    #oProper.wDigital_Inputs := #PI.wDigital_Inputs;
	    
	    //Mapping the signals of the control word:
	    #PO.x_Bit_0_Enable_Emergency_Stop := #IProper.x_Bit_0_Enable_Emergency_Stop;
	    #PO.x_Bit_1_Enable_Application_Stop := #IProper.x_Bit_1_Enable_Application_Stop;
	    #PO.x_Bit_4_Jog_positive := #IProper.x_Bit_4_Jog_positive;
	    #PO.x_Bit_5_Jog_negative := #IProper.x_Bit_5_Jog_negative;
	    #PO.x_Bit_3_Release_Brake := #IProper.x_Bit_3_Release_Brake;
	    #PO.x_Bit_7_Start_Stop := #IProper.x_Bit_7_Start_Stop;
	    #PO.x_Bit_8_Fault_Reset := #IProper.x_Bit_8_Fault_Reset;
	    #PO.x_Bit_10_Activate_DriveTrain2 := #IProper.x_Bit_10_Activate_DriveTrain2;
	    #PO.x_Bit_13_Activate_Output_Stage_Inhibit := #IProper.x_Bit_13_Activate_Output_Stage_Inhibit;
	    #PO.x_Bit_14_Activate_StandBy_Mode := #IProper.x_Bit_14_Activate_StandBy_Mode;
	    #PO.x_Bit_15_Heartbeat_IN := #IProper.x_Bit_15_Heartbeat_IN;
	    
	    //Set the not used Bits to "false"
	    #PO.x_Bit_2_Reserved:= FALSE;
	    #PO.x_Bit_6_Apply_relative_Position := FALSE;
	    #PO.x_Bit_9_Reserved := FALSE;
	    #PO.x_Bit_11_Reserved := FALSE;
	    #PO.x_Bit_12_Deactivate_SW_Limit_switches := false;
	    
	    //Assig the POs 2..5
	    #PO.iSetpoint_Speed := #IProper.iSetpoint_Speed;
	    #PO.iSetpoint_Acceleration := #IProper.iSetpoint_Acceleration;
	    #PO.iSetpoint_Deceleration := #IProper.iSetpoint_Deceleration;
	    #PO.wDigital_Outputs := #IProper.wDigital_Outputs;
	    
	ELSE
	    GOTO END;
	END_IF;
	
	//DPWR_DAT: Write consistent data of a DP standard slave/PROFINET IO device
	#DPWR_RET_VAL := DPWR_DAT(LADDR := #HW_IDENTIFIER, RECORD := #PO);
	
	END:
	IF #DPRD_RET_VAL <> 0 OR #DPWR_RET_VAL <> 0 THEN
	    #COMMUNICATION_OK := FALSE;
	    //Erase FC outputs in case of an error
	    #oProper.x_Bit_0_Ready := FALSE;
	    #oProper.x_Bit_1_STO_inactive := FALSE;
	    #oProper.x_Bit_2_Output_Stage_enabled := FALSE;
	    #oProper.x_Bit_3_Brake_released := FALSE;
	    #oProper.x_Bit_4_Motor_turning := FALSE;
	    #oProper.x_Bit_8_Fault := FALSE;
	    #oProper.x_Bit_9_Warning := FALSE;
	    #oProper.x_Bit_10_DriveTrain2_active := FALSE;
	    #oProper.x_Bit_11_Setp_actual_speed_comp_signal_active := FALSE;
	    #oProper.x_Bit_14_StandBy_Mode_active := FALSE;
	    #oProper.x_Bit_15_Heartbeat_OUT := FALSE;
	    #oProper.iActual_Speed := 0;
	    #oProper.wStatus_main_fault_sub_fault := 0;
	    #oProper.iActual_Torque := 0;
	    #oProper.wDigital_Inputs := 0;
	END_IF;
END_FUNCTION

FUNCTION_BLOCK "Pallet_Transport_Row_4"   // FB14, LAD
{ S7_Optimized_Access := 'TRUE' }
// stored: MemoryReserve 100, SetENOAutomatically false
   VAR_INPUT
      Start_Station : "Station";
      Destination_Station : "Station";
      Reverse_Rotation : Bool;
      iButton_StS_StD : Bool;
      iButton_StD_StS : Bool;
      isEndingStation_STD : Bool;
      isEndingStation_STS : Bool;
      TandemOperation : Bool;
      TandemSpeed : Int;
   END_VAR
   VAR_OUTPUT
      oButton_StS_StD_LED : Bool;
      oStatus_HMI_StS_StD : Bool;
      oStatus_HMI_StD_StS : Bool;
      oCentering : Bool;
      Stop_Drive_Button : Bool;
      Stop_Drive_HMI : Bool;
      Centering_Alarm : Bool;
   END_VAR
   VAR_IN_OUT
      iDriveStS_Param : "SEW_MOVIKIT_VelocityDrive_SETPOINTS_V2.1";
      oDriveStS_Param : "SEW_MOVIKIT_VelocityDrive_STATUS_V2.1";
      iDriveStD_Param : "SEW_MOVIKIT_VelocityDrive_SETPOINTS_V2.1";
      oDriveStD_Param : "SEW_MOVIKIT_VelocityDrive_STATUS_V2.1";
      iDriveStS_double_Param : "SEW_MOVIKIT_VelocityDrive_SETPOINTS_V2.1";
      oDriveStS_double_Param : "SEW_MOVIKIT_VelocityDrive_STATUS_V2.1";
      iDriveStD_double_Param : "SEW_MOVIKIT_VelocityDrive_SETPOINTS_V2.1";
      oDriveStD_double_Param : "SEW_MOVIKIT_VelocityDrive_STATUS_V2.1";
      isCentering : Bool;
      HMI_StS_StD : Bool;
      HMI_StD_StS : Bool;
   END_VAR
   VAR
      Drive_To_Destination : Bool;
      Set_Speed : Int;
      Set_Speed_Reverse : Int;
      CommunicationOk : Bool;
      Jog_StS : Bool;
      Jog_StD : Bool;
      CenteringStep : Int;
      TON_Centering : TON_TIME;
      trigTimeout { S7_SetPoint := 'True'} : R_TRIG;
      Trig_StS_StD { S7_SetPoint := 'True'} : Bool;
      Trig_StD_StS : Bool;
      Reset_StS_StD : Bool;
      Reset_StD_StS : Bool;
      Timer_Drive_Error_Button : TON_TIME;
      Timer_Drive_Error_HMI : TON_TIME;
      STOP_DRIVERS { S7_SetPoint := 'True'} : Bool;
   END_VAR
   VAR_TEMP
      LED_StD_STS : Bool;
      LED_StS_STD : Bool;
   END_VAR
   VAR CONSTANT
      ACC : Int := 300;
      DCC : Int := 400;
      SPEED_BACK : Int := -100;
      SPEED_FWD : Int := 100;
   END_VAR
   VAR_TEMP   // added for the SCL form of the ladder/FBD networks
      _w1 : Bool;
      _w2 : Bool;
      _w3 : Bool;
      _w4 : Bool;
   END_VAR
BEGIN

REGION Network 1: Reset commands
